REGION Network 67: FAT Mode All Check
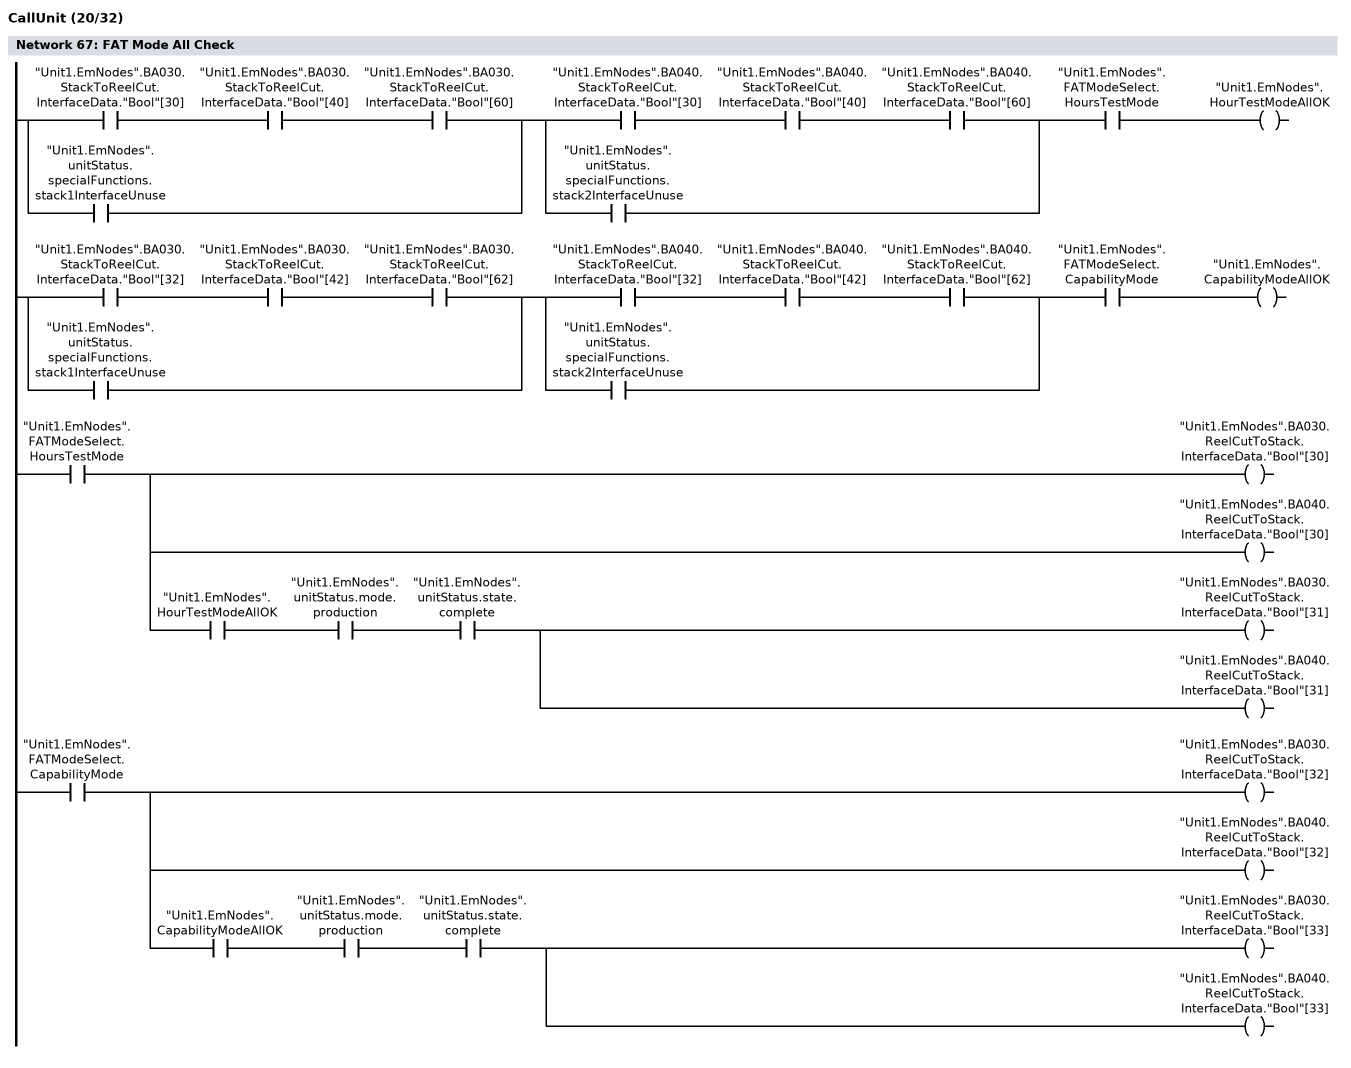
   RUNG wire#powerrail
      Contact( "Unit1.EmNodes".BA030.StackToReelCut.InterfaceData."Bool"[30] )
      Contact( "Unit1.EmNodes".BA030.StackToReelCut.InterfaceData."Bool"[40] )
      Contact( "Unit1.EmNodes".BA030.StackToReelCut.InterfaceData."Bool"[60] )
      wire#w1
      Contact( "Unit1.EmNodes".BA040.StackToReelCut.InterfaceData."Bool"[30] )
      Contact( "Unit1.EmNodes".BA040.StackToReelCut.InterfaceData."Bool"[40] )
      Contact( "Unit1.EmNodes".BA040.StackToReelCut.InterfaceData."Bool"[60] )
      wire#w2
      Contact( "Unit1.EmNodes".FATModeSelect.HoursTestMode )
      Coil( "Unit1.EmNodes".HourTestModeAllOK )
   END_RUNG
   RUNG wire#powerrail
      Contact( "Unit1.EmNodes".unitStatus.specialFunctions.stack1InterfaceUnuse )
   END_RUNG wire#w1
   RUNG wire#w1
      Contact( "Unit1.EmNodes".unitStatus.specialFunctions.stack2InterfaceUnuse )
   END_RUNG wire#w2
   RUNG wire#powerrail
      Contact( "Unit1.EmNodes".BA030.StackToReelCut.InterfaceData."Bool"[32] )
      Contact( "Unit1.EmNodes".BA030.StackToReelCut.InterfaceData."Bool"[42] )
      Contact( "Unit1.EmNodes".BA030.StackToReelCut.InterfaceData."Bool"[62] )
      wire#w3
      Contact( "Unit1.EmNodes".BA040.StackToReelCut.InterfaceData."Bool"[32] )
      Contact( "Unit1.EmNodes".BA040.StackToReelCut.InterfaceData."Bool"[42] )
      Contact( "Unit1.EmNodes".BA040.StackToReelCut.InterfaceData."Bool"[62] )
      wire#w4
      Contact( "Unit1.EmNodes".FATModeSelect.CapabilityMode )
      Coil( "Unit1.EmNodes".CapabilityModeAllOK )
   END_RUNG
   RUNG wire#powerrail
      Contact( "Unit1.EmNodes".unitStatus.specialFunctions.stack1InterfaceUnuse )
   END_RUNG wire#w3
   RUNG wire#w3
      Contact( "Unit1.EmNodes".unitStatus.specialFunctions.stack2InterfaceUnuse )
   END_RUNG wire#w4
   RUNG wire#powerrail
      Contact( "Unit1.EmNodes".FATModeSelect.HoursTestMode )
      wire#w5
      Coil( "Unit1.EmNodes".BA030.ReelCutToStack.InterfaceData."Bool"[30] )
   END_RUNG
   RUNG wire#w5
      Coil( "Unit1.EmNodes".BA040.ReelCutToStack.InterfaceData."Bool"[30] )
   END_RUNG
   RUNG wire#w5
      Contact( "Unit1.EmNodes".HourTestModeAllOK )
      Contact( "Unit1.EmNodes".unitStatus.mode.production )
      Contact( "Unit1.EmNodes".unitStatus.state.complete )
      wire#w6
      Coil( "Unit1.EmNodes".BA030.ReelCutToStack.InterfaceData."Bool"[31] )
   END_RUNG
   RUNG wire#w6
      Coil( "Unit1.EmNodes".BA040.ReelCutToStack.InterfaceData."Bool"[31] )
   END_RUNG
   RUNG wire#powerrail
      Contact( "Unit1.EmNodes".FATModeSelect.CapabilityMode )
      wire#w7
      Coil( "Unit1.EmNodes".BA030.ReelCutToStack.InterfaceData."Bool"[32] )
   END_RUNG
   RUNG wire#w7
      Coil( "Unit1.EmNodes".BA040.ReelCutToStack.InterfaceData."Bool"[32] )
   END_RUNG
   RUNG wire#w7
      Contact( "Unit1.EmNodes".CapabilityModeAllOK )
      Contact( "Unit1.EmNodes".unitStatus.mode.production )
      Contact( "Unit1.EmNodes".unitStatus.state.complete )
      wire#w8
      Coil( "Unit1.EmNodes".BA030.ReelCutToStack.InterfaceData."Bool"[33] )
   END_RUNG
   RUNG wire#w8
      Coil( "Unit1.EmNodes".BA040.ReelCutToStack.InterfaceData."Bool"[33] )
   END_RUNG
   // the same network as SCL:
   "Unit1.EmNodes".HourTestModeAllOK := (("Unit1.EmNodes".BA030.StackToReelCut.InterfaceData."Bool"[30] AND "Unit1.EmNodes".BA030.StackToReelCut.InterfaceData."Bool"[40] AND "Unit1.EmNodes".BA030.StackToReelCut.InterfaceData."Bool"[60]) OR "Unit1.EmNodes".unitStatus.specialFunctions.stack1InterfaceUnuse) AND (("Unit1.EmNodes".BA040.StackToReelCut.InterfaceData."Bool"[30] AND "Unit1.EmNodes".BA040.StackToReelCut.InterfaceData."Bool"[40] AND "Unit1.EmNodes".BA040.StackToReelCut.InterfaceData."Bool"[60]) OR "Unit1.EmNodes".unitStatus.specialFunctions.stack2InterfaceUnuse) AND "Unit1.EmNodes".FATModeSelect.HoursTestMode;
   "Unit1.EmNodes".CapabilityModeAllOK := (("Unit1.EmNodes".BA030.StackToReelCut.InterfaceData."Bool"[32] AND "Unit1.EmNodes".BA030.StackToReelCut.InterfaceData."Bool"[42] AND "Unit1.EmNodes".BA030.StackToReelCut.InterfaceData."Bool"[62]) OR "Unit1.EmNodes".unitStatus.specialFunctions.stack1InterfaceUnuse) AND (("Unit1.EmNodes".BA040.StackToReelCut.InterfaceData."Bool"[32] AND "Unit1.EmNodes".BA040.StackToReelCut.InterfaceData."Bool"[42] AND "Unit1.EmNodes".BA040.StackToReelCut.InterfaceData."Bool"[62]) OR "Unit1.EmNodes".unitStatus.specialFunctions.stack2InterfaceUnuse) AND "Unit1.EmNodes".FATModeSelect.CapabilityMode;
   "Unit1.EmNodes".BA030.ReelCutToStack.InterfaceData."Bool"[30] := "Unit1.EmNodes".FATModeSelect.HoursTestMode;
   "Unit1.EmNodes".BA040.ReelCutToStack.InterfaceData."Bool"[30] := "Unit1.EmNodes".FATModeSelect.HoursTestMode;
   "Unit1.EmNodes".BA030.ReelCutToStack.InterfaceData."Bool"[31] := "Unit1.EmNodes".FATModeSelect.HoursTestMode AND "Unit1.EmNodes".HourTestModeAllOK AND "Unit1.EmNodes".unitStatus.mode.production AND "Unit1.EmNodes".unitStatus.state.complete;
   "Unit1.EmNodes".BA040.ReelCutToStack.InterfaceData."Bool"[31] := "Unit1.EmNodes".FATModeSelect.HoursTestMode AND "Unit1.EmNodes".HourTestModeAllOK AND "Unit1.EmNodes".unitStatus.mode.production AND "Unit1.EmNodes".unitStatus.state.complete;
   "Unit1.EmNodes".BA030.ReelCutToStack.InterfaceData."Bool"[32] := "Unit1.EmNodes".FATModeSelect.CapabilityMode;
   "Unit1.EmNodes".BA040.ReelCutToStack.InterfaceData."Bool"[32] := "Unit1.EmNodes".FATModeSelect.CapabilityMode;
   "Unit1.EmNodes".BA030.ReelCutToStack.InterfaceData."Bool"[33] := "Unit1.EmNodes".FATModeSelect.CapabilityMode AND "Unit1.EmNodes".CapabilityModeAllOK AND "Unit1.EmNodes".unitStatus.mode.production AND "Unit1.EmNodes".unitStatus.state.complete;
   "Unit1.EmNodes".BA040.ReelCutToStack.InterfaceData."Bool"[33] := "Unit1.EmNodes".FATModeSelect.CapabilityMode AND "Unit1.EmNodes".CapabilityModeAllOK AND "Unit1.EmNodes".unitStatus.mode.production AND "Unit1.EmNodes".unitStatus.state.complete;
END_REGION

REGION Network 68: HoursTest Mode
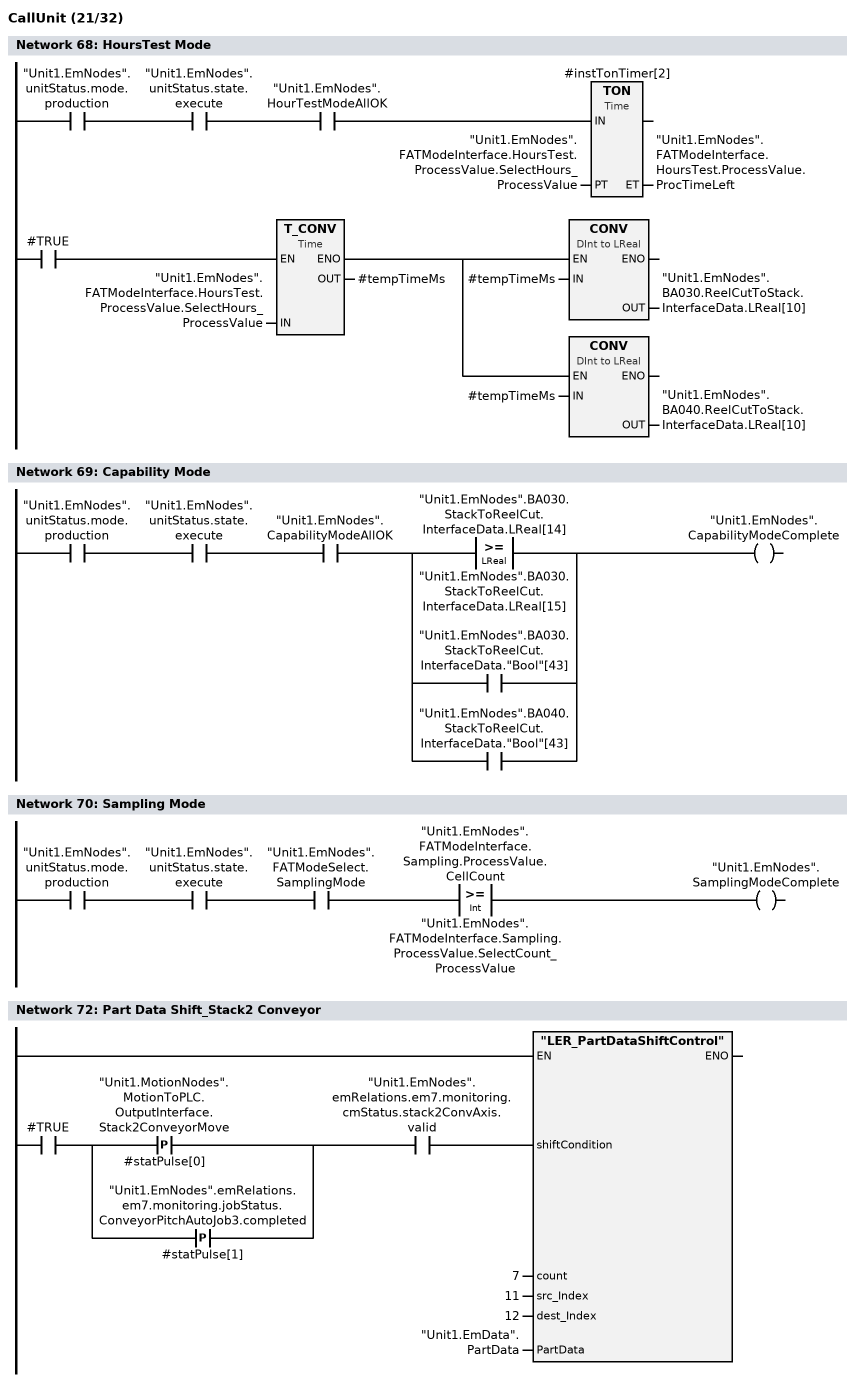
   RUNG wire#powerrail
      Contact( "Unit1.EmNodes".unitStatus.mode.production )
      Contact( "Unit1.EmNodes".unitStatus.state.execute )
      Contact( "Unit1.EmNodes".HourTestModeAllOK )
      { S7_Templates := "time_type := Time" } #instTonTimer[2].TON(pt := "Unit1.EmNodes".FATModeInterface.HoursTest.ProcessValue.SelectHours_ProcessValue, et => "Unit1.EmNodes".FATModeInterface.HoursTest.ProcessValue.ProcTimeLeft)
   END_RUNG
   RUNG wire#powerrail
      Contact( #TRUE )
      { S7_Templates := "[src_type := Time, dest_type := DInt]" } T_CONV(IN := "Unit1.EmNodes".FATModeInterface.HoursTest.ProcessValue.SelectHours_ProcessValue, OUT => #tempTimeMs)
      wire#w1
      { S7_Templates := "[SrcType := DInt, DestType := LReal]" } Convert(in := #tempTimeMs, out => "Unit1.EmNodes".BA030.ReelCutToStack.InterfaceData.LReal[10])
   END_RUNG
   RUNG wire#w1
      { S7_Templates := "[SrcType := DInt, DestType := LReal]" } Convert(in := #tempTimeMs, out => "Unit1.EmNodes".BA040.ReelCutToStack.InterfaceData.LReal[10])
   END_RUNG
   // the same network as SCL:
   #instTonTimer[2].TON(IN := "Unit1.EmNodes".unitStatus.mode.production AND "Unit1.EmNodes".unitStatus.state.execute AND "Unit1.EmNodes".HourTestModeAllOK,
                        PT := "Unit1.EmNodes".FATModeInterface.HoursTest.ProcessValue.SelectHours_ProcessValue,
                        ET => "Unit1.EmNodes".FATModeInterface.HoursTest.ProcessValue.ProcTimeLeft);
   T_CONV(EN := #TRUE,
          IN := "Unit1.EmNodes".FATModeInterface.HoursTest.ProcessValue.SelectHours_ProcessValue,
          OUT => #tempTimeMs,
          ENO => #_w1);
   IF #_w1 THEN
       "Unit1.EmNodes".BA030.ReelCutToStack.InterfaceData.LReal[10] := DINT_TO_LREAL(#tempTimeMs);
       "Unit1.EmNodes".BA040.ReelCutToStack.InterfaceData.LReal[10] := DINT_TO_LREAL(#tempTimeMs);
   END_IF;
END_REGION

REGION Network 69: Capability Mode
   RUNG wire#powerrail
      Contact( "Unit1.EmNodes".unitStatus.mode.production )
      Contact( "Unit1.EmNodes".unitStatus.state.execute )
      Contact( "Unit1.EmNodes".CapabilityModeAllOK )
      wire#w1
      { S7_Templates := "SrcType := LReal" } GE_Contact(in1 := "Unit1.EmNodes".BA030.StackToReelCut.InterfaceData.LReal[14], in2 := "Unit1.EmNodes".BA030.StackToReelCut.InterfaceData.LReal[15])
      wire#w2
      Coil( "Unit1.EmNodes".CapabilityModeComplete )
   END_RUNG
   RUNG wire#w1
      Contact( "Unit1.EmNodes".BA030.StackToReelCut.InterfaceData."Bool"[43] )
   END_RUNG wire#w2
   RUNG wire#w1
      Contact( "Unit1.EmNodes".BA040.StackToReelCut.InterfaceData."Bool"[43] )
   END_RUNG wire#w2
   // the same network as SCL:
   "Unit1.EmNodes".CapabilityModeComplete := "Unit1.EmNodes".unitStatus.mode.production AND "Unit1.EmNodes".unitStatus.state.execute AND "Unit1.EmNodes".CapabilityModeAllOK AND (("Unit1.EmNodes".BA030.StackToReelCut.InterfaceData.LReal[14] >= "Unit1.EmNodes".BA030.StackToReelCut.InterfaceData.LReal[15]) OR "Unit1.EmNodes".BA030.StackToReelCut.InterfaceData."Bool"[43] OR "Unit1.EmNodes".BA040.StackToReelCut.InterfaceData."Bool"[43]);
END_REGION

REGION Network 70: Sampling Mode
   RUNG wire#powerrail
      Contact( "Unit1.EmNodes".unitStatus.mode.production )
      Contact( "Unit1.EmNodes".unitStatus.state.execute )
      Contact( "Unit1.EmNodes".FATModeSelect.SamplingMode )
      { S7_Templates := "SrcType := Int" } GE_Contact(in1 := "Unit1.EmNodes".FATModeInterface.Sampling.ProcessValue.CellCount, in2 := "Unit1.EmNodes".FATModeInterface.Sampling.ProcessValue.SelectCount_ProcessValue)
      Coil( "Unit1.EmNodes".SamplingModeComplete )
   END_RUNG
   // the same network as SCL:
   "Unit1.EmNodes".SamplingModeComplete := "Unit1.EmNodes".unitStatus.mode.production AND "Unit1.EmNodes".unitStatus.state.execute AND "Unit1.EmNodes".FATModeSelect.SamplingMode AND ("Unit1.EmNodes".FATModeInterface.Sampling.ProcessValue.CellCount >= "Unit1.EmNodes".FATModeInterface.Sampling.ProcessValue.SelectCount_ProcessValue);
END_REGION

REGION Network 71: ******************** Part Data Shift ********************
END_REGION

REGION Network 72: Part Data Shift_Stack2 Conveyor
   RUNG wire#powerrail
      "LER_PartDataShiftControl"(shiftCondition := wire#w3, count := 7, src_Index := 11, dest_Index := 12, PartData := "Unit1.EmData".PartData)
   END_RUNG
   RUNG wire#powerrail
      Contact( #TRUE )
      wire#w1
      P_Contact(operand := "Unit1.MotionNodes".MotionToPLC.OutputInterface.Stack2ConveyorMove, bit := #statPulse[0])
      wire#w2
      Contact( "Unit1.EmNodes".emRelations.em7.monitoring.cmStatus.stack2ConvAxis.valid )
   END_RUNG wire#w3
   RUNG wire#w1
      P_Contact(operand := "Unit1.EmNodes".emRelations.em7.monitoring.jobStatus.ConveyorPitchAutoJob3.completed, bit := #statPulse[1])
   END_RUNG wire#w2
   // the same network as SCL:
   #_w1 := #TRUE AND "Unit1.MotionNodes".MotionToPLC.OutputInterface.Stack2ConveyorMove AND NOT #statPulse[0];   // rising edge of "Unit1.MotionNodes".MotionToPLC.OutputInterface.Stack2ConveyorMove
   #statPulse[0] := "Unit1.MotionNodes".MotionToPLC.OutputInterface.Stack2ConveyorMove;
   #_w2 := #TRUE AND "Unit1.EmNodes".emRelations.em7.monitoring.jobStatus.ConveyorPitchAutoJob3.completed AND NOT #statPulse[1];   // rising edge of "Unit1.EmNodes".emRelations.em7.monitoring.jobStatus.ConveyorPitchAutoJob3.completed
   #statPulse[1] := "Unit1.EmNodes".emRelations.em7.monitoring.jobStatus.ConveyorPitchAutoJob3.completed;
   "LER_PartDataShiftControl"(shiftCondition := (#_w1 OR #_w2) AND "Unit1.EmNodes".emRelations.em7.monitoring.cmStatus.stack2ConvAxis.valid,
                           count := 7,
                           src_Index := 11,
                           dest_Index := 12,
                           PartData := "Unit1.EmData".PartData);
END_REGION

REGION Network 73: Part Data Shift_Stack1 Conveyor
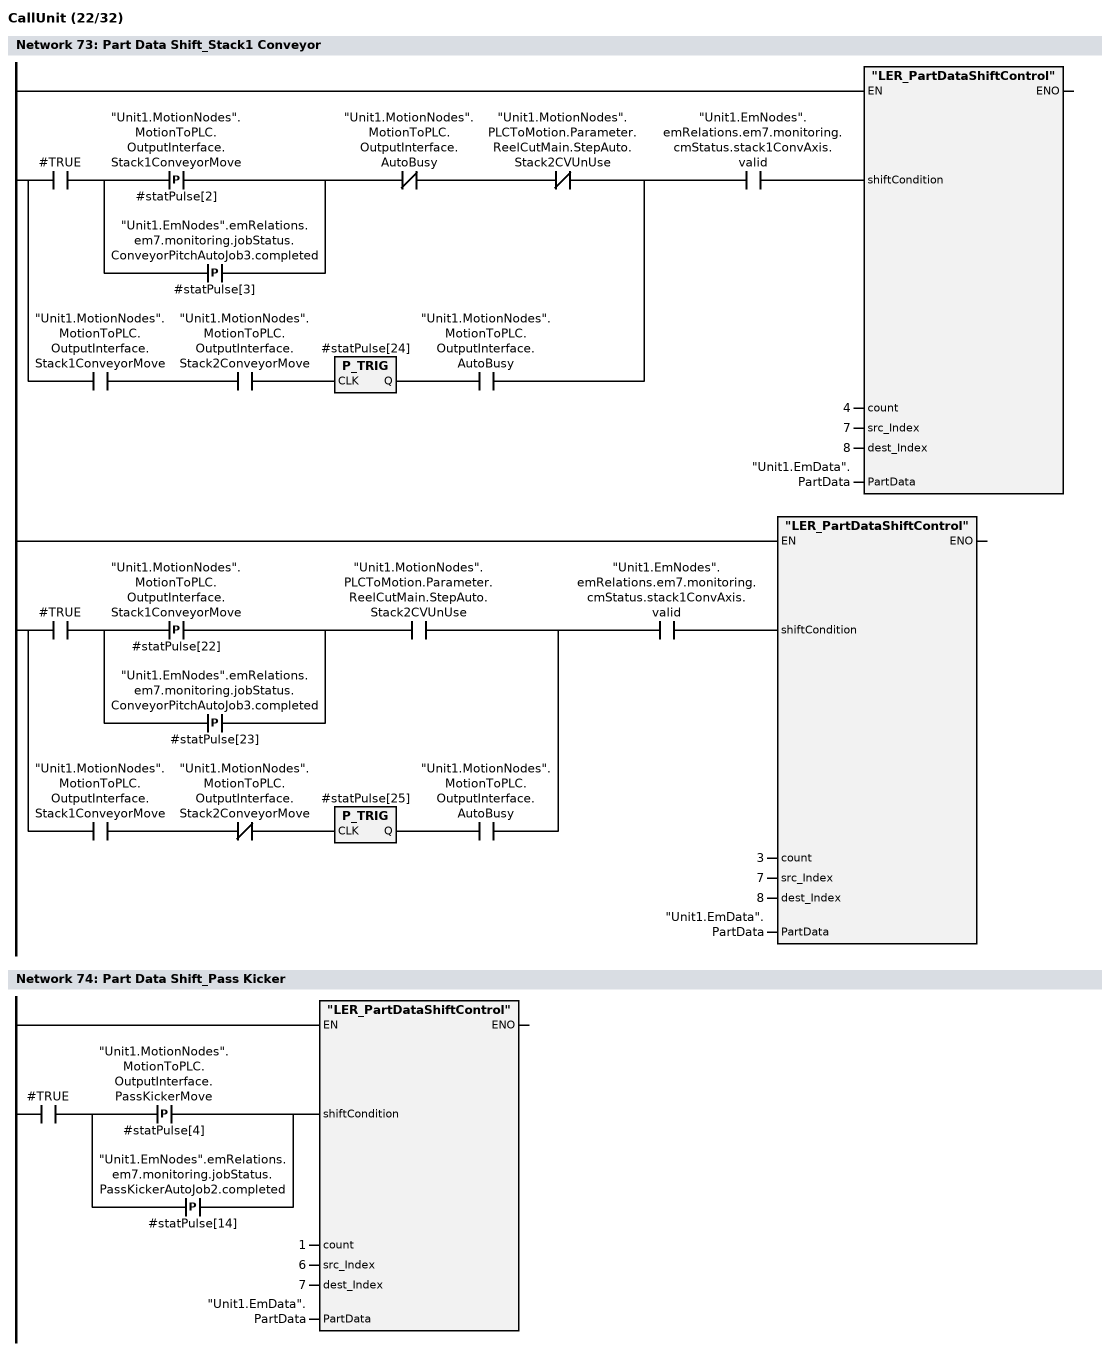
   RUNG wire#powerrail
      "LER_PartDataShiftControl"(shiftCondition := wire#w4, count := 4, src_Index := 7, dest_Index := 8, PartData := "Unit1.EmData".PartData)
   END_RUNG
   RUNG wire#powerrail
      Contact( #TRUE )
      wire#w1
      P_Contact(operand := "Unit1.MotionNodes".MotionToPLC.OutputInterface.Stack1ConveyorMove, bit := #statPulse[2])
      wire#w2
      I_Contact( "Unit1.MotionNodes".MotionToPLC.OutputInterface.AutoBusy )
      I_Contact( "Unit1.MotionNodes".PLCToMotion.Parameter.ReelCutMain.StepAuto.Stack2CVUnUse )
      wire#w3
      Contact( "Unit1.EmNodes".emRelations.em7.monitoring.cmStatus.stack1ConvAxis.valid )
   END_RUNG wire#w4
   RUNG wire#w1
      P_Contact(operand := "Unit1.EmNodes".emRelations.em7.monitoring.jobStatus.ConveyorPitchAutoJob3.completed, bit := #statPulse[3])
   END_RUNG wire#w2
   RUNG wire#powerrail
      Contact( "Unit1.MotionNodes".MotionToPLC.OutputInterface.Stack1ConveyorMove )
      Contact( "Unit1.MotionNodes".MotionToPLC.OutputInterface.Stack2ConveyorMove )
      P_Trig( #statPulse[24] )
      Contact( "Unit1.MotionNodes".MotionToPLC.OutputInterface.AutoBusy )
   END_RUNG wire#w3
   RUNG wire#powerrail
      "LER_PartDataShiftControl"(shiftCondition := wire#w8, count := 3, src_Index := 7, dest_Index := 8, PartData := "Unit1.EmData".PartData)
   END_RUNG
   RUNG wire#powerrail
      Contact( #TRUE )
      wire#w5
      P_Contact(operand := "Unit1.MotionNodes".MotionToPLC.OutputInterface.Stack1ConveyorMove, bit := #statPulse[22])
      wire#w6
      Contact( "Unit1.MotionNodes".PLCToMotion.Parameter.ReelCutMain.StepAuto.Stack2CVUnUse )
      wire#w7
      Contact( "Unit1.EmNodes".emRelations.em7.monitoring.cmStatus.stack1ConvAxis.valid )
   END_RUNG wire#w8
   RUNG wire#w5
      P_Contact(operand := "Unit1.EmNodes".emRelations.em7.monitoring.jobStatus.ConveyorPitchAutoJob3.completed, bit := #statPulse[23])
   END_RUNG wire#w6
   RUNG wire#powerrail
      Contact( "Unit1.MotionNodes".MotionToPLC.OutputInterface.Stack1ConveyorMove )
      I_Contact( "Unit1.MotionNodes".MotionToPLC.OutputInterface.Stack2ConveyorMove )
      P_Trig( #statPulse[25] )
      Contact( "Unit1.MotionNodes".MotionToPLC.OutputInterface.AutoBusy )
   END_RUNG wire#w7
   // the same network as SCL:
   #_w1 := #TRUE AND "Unit1.MotionNodes".MotionToPLC.OutputInterface.Stack1ConveyorMove AND NOT #statPulse[2];   // rising edge of "Unit1.MotionNodes".MotionToPLC.OutputInterface.Stack1ConveyorMove
   #statPulse[2] := "Unit1.MotionNodes".MotionToPLC.OutputInterface.Stack1ConveyorMove;
   #_w2 := #TRUE AND "Unit1.EmNodes".emRelations.em7.monitoring.jobStatus.ConveyorPitchAutoJob3.completed AND NOT #statPulse[3];   // rising edge of "Unit1.EmNodes".emRelations.em7.monitoring.jobStatus.ConveyorPitchAutoJob3.completed
   #statPulse[3] := "Unit1.EmNodes".emRelations.em7.monitoring.jobStatus.ConveyorPitchAutoJob3.completed;
   #_w3 := "Unit1.MotionNodes".MotionToPLC.OutputInterface.Stack1ConveyorMove AND "Unit1.MotionNodes".MotionToPLC.OutputInterface.Stack2ConveyorMove;
   #_w4 := #_w3 AND NOT #statPulse[24];   // rising edge
   #statPulse[24] := #_w3;
   "LER_PartDataShiftControl"(shiftCondition := (((#_w1 OR #_w2) AND NOT "Unit1.MotionNodes".MotionToPLC.OutputInterface.AutoBusy AND NOT "Unit1.MotionNodes".PLCToMotion.Parameter.ReelCutMain.StepAuto.Stack2CVUnUse) OR (#_w4 AND "Unit1.MotionNodes".MotionToPLC.OutputInterface.AutoBusy)) AND "Unit1.EmNodes".emRelations.em7.monitoring.cmStatus.stack1ConvAxis.valid,
                           count := 4,
                           src_Index := 7,
                           dest_Index := 8,
                           PartData := "Unit1.EmData".PartData);
   #_w5 := #TRUE AND "Unit1.MotionNodes".MotionToPLC.OutputInterface.Stack1ConveyorMove AND NOT #statPulse[22];   // rising edge of "Unit1.MotionNodes".MotionToPLC.OutputInterface.Stack1ConveyorMove
   #statPulse[22] := "Unit1.MotionNodes".MotionToPLC.OutputInterface.Stack1ConveyorMove;
   #_w6 := #TRUE AND "Unit1.EmNodes".emRelations.em7.monitoring.jobStatus.ConveyorPitchAutoJob3.completed AND NOT #statPulse[23];   // rising edge of "Unit1.EmNodes".emRelations.em7.monitoring.jobStatus.ConveyorPitchAutoJob3.completed
   #statPulse[23] := "Unit1.EmNodes".emRelations.em7.monitoring.jobStatus.ConveyorPitchAutoJob3.completed;
   #_w7 := "Unit1.MotionNodes".MotionToPLC.OutputInterface.Stack1ConveyorMove AND NOT "Unit1.MotionNodes".MotionToPLC.OutputInterface.Stack2ConveyorMove;
   #_w8 := #_w7 AND NOT #statPulse[25];   // rising edge
   #statPulse[25] := #_w7;
   "LER_PartDataShiftControl"(shiftCondition := (((#_w5 OR #_w6) AND "Unit1.MotionNodes".PLCToMotion.Parameter.ReelCutMain.StepAuto.Stack2CVUnUse) OR (#_w8 AND "Unit1.MotionNodes".MotionToPLC.OutputInterface.AutoBusy)) AND "Unit1.EmNodes".emRelations.em7.monitoring.cmStatus.stack1ConvAxis.valid,
                           count := 3,
                           src_Index := 7,
                           dest_Index := 8,
                           PartData := "Unit1.EmData".PartData);
END_REGION

REGION Network 74: Part Data Shift_Pass Kicker
   RUNG wire#powerrail
      "LER_PartDataShiftControl"(shiftCondition := wire#w2, count := 1, src_Index := 6, dest_Index := 7, PartData := "Unit1.EmData".PartData)
   END_RUNG
   RUNG wire#powerrail
      Contact( #TRUE )
      wire#w1
      P_Contact(operand := "Unit1.MotionNodes".MotionToPLC.OutputInterface.PassKickerMove, bit := #statPulse[4])
   END_RUNG wire#w2
   RUNG wire#w1
      P_Contact(operand := "Unit1.EmNodes".emRelations.em7.monitoring.jobStatus.PassKickerAutoJob2.completed, bit := #statPulse[14])
   END_RUNG wire#w2
   // the same network as SCL:
   #_w1 := #TRUE AND "Unit1.MotionNodes".MotionToPLC.OutputInterface.PassKickerMove AND NOT #statPulse[4];   // rising edge of "Unit1.MotionNodes".MotionToPLC.OutputInterface.PassKickerMove
   #statPulse[4] := "Unit1.MotionNodes".MotionToPLC.OutputInterface.PassKickerMove;
   #_w2 := #TRUE AND "Unit1.EmNodes".emRelations.em7.monitoring.jobStatus.PassKickerAutoJob2.completed AND NOT #statPulse[14];   // rising edge of "Unit1.EmNodes".emRelations.em7.monitoring.jobStatus.PassKickerAutoJob2.completed
   #statPulse[14] := "Unit1.EmNodes".emRelations.em7.monitoring.jobStatus.PassKickerAutoJob2.completed;
   "LER_PartDataShiftControl"(shiftCondition := #_w1 OR #_w2,
                           count := 1,
                           src_Index := 6,
                           dest_Index := 7,
                           PartData := "Unit1.EmData".PartData);
END_REGION

REGION Network 75: Part Data Shift_NG Kicker
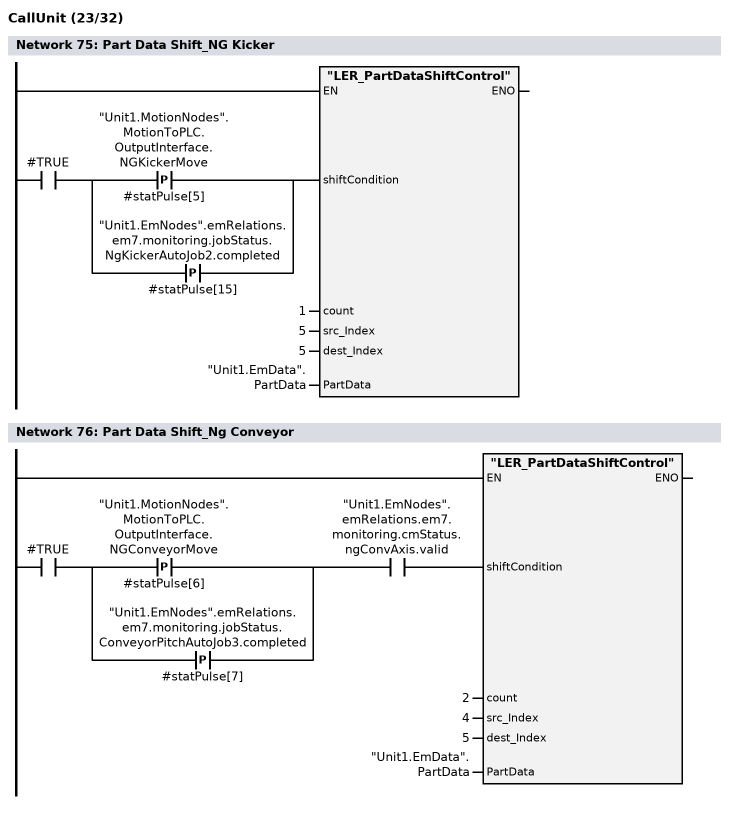
   RUNG wire#powerrail
      "LER_PartDataShiftControl"(shiftCondition := wire#w2, count := 1, src_Index := 5, dest_Index := 5, PartData := "Unit1.EmData".PartData)
   END_RUNG
   RUNG wire#powerrail
      Contact( #TRUE )
      wire#w1
      P_Contact(operand := "Unit1.MotionNodes".MotionToPLC.OutputInterface.NGKickerMove, bit := #statPulse[5])
   END_RUNG wire#w2
   RUNG wire#w1
      P_Contact(operand := "Unit1.EmNodes".emRelations.em7.monitoring.jobStatus.NgKickerAutoJob2.completed, bit := #statPulse[15])
   END_RUNG wire#w2
   // the same network as SCL:
   #_w1 := #TRUE AND "Unit1.MotionNodes".MotionToPLC.OutputInterface.NGKickerMove AND NOT #statPulse[5];   // rising edge of "Unit1.MotionNodes".MotionToPLC.OutputInterface.NGKickerMove
   #statPulse[5] := "Unit1.MotionNodes".MotionToPLC.OutputInterface.NGKickerMove;
   #_w2 := #TRUE AND "Unit1.EmNodes".emRelations.em7.monitoring.jobStatus.NgKickerAutoJob2.completed AND NOT #statPulse[15];   // rising edge of "Unit1.EmNodes".emRelations.em7.monitoring.jobStatus.NgKickerAutoJob2.completed
   #statPulse[15] := "Unit1.EmNodes".emRelations.em7.monitoring.jobStatus.NgKickerAutoJob2.completed;
   "LER_PartDataShiftControl"(shiftCondition := #_w1 OR #_w2,
                           count := 1,
                           src_Index := 5,
                           dest_Index := 5,
                           PartData := "Unit1.EmData".PartData);
END_REGION

REGION Network 76: Part Data Shift_Ng Conveyor
   RUNG wire#powerrail
      "LER_PartDataShiftControl"(shiftCondition := wire#w3, count := 2, src_Index := 4, dest_Index := 5, PartData := "Unit1.EmData".PartData)
   END_RUNG
   RUNG wire#powerrail
      Contact( #TRUE )
      wire#w1
      P_Contact(operand := "Unit1.MotionNodes".MotionToPLC.OutputInterface.NGConveyorMove, bit := #statPulse[6])
      wire#w2
      Contact( "Unit1.EmNodes".emRelations.em7.monitoring.cmStatus.ngConvAxis.valid )
   END_RUNG wire#w3
   RUNG wire#w1
      P_Contact(operand := "Unit1.EmNodes".emRelations.em7.monitoring.jobStatus.ConveyorPitchAutoJob3.completed, bit := #statPulse[7])
   END_RUNG wire#w2
   // the same network as SCL:
   #_w1 := #TRUE AND "Unit1.MotionNodes".MotionToPLC.OutputInterface.NGConveyorMove AND NOT #statPulse[6];   // rising edge of "Unit1.MotionNodes".MotionToPLC.OutputInterface.NGConveyorMove
   #statPulse[6] := "Unit1.MotionNodes".MotionToPLC.OutputInterface.NGConveyorMove;
   #_w2 := #TRUE AND "Unit1.EmNodes".emRelations.em7.monitoring.jobStatus.ConveyorPitchAutoJob3.completed AND NOT #statPulse[7];   // rising edge of "Unit1.EmNodes".emRelations.em7.monitoring.jobStatus.ConveyorPitchAutoJob3.completed
   #statPulse[7] := "Unit1.EmNodes".emRelations.em7.monitoring.jobStatus.ConveyorPitchAutoJob3.completed;
   "LER_PartDataShiftControl"(shiftCondition := (#_w1 OR #_w2) AND "Unit1.EmNodes".emRelations.em7.monitoring.cmStatus.ngConvAxis.valid,
                           count := 2,
                           src_Index := 4,
                           dest_Index := 5,
                           PartData := "Unit1.EmData".PartData);
END_REGION

REGION Network 77: Part Data Shift_Cut Conveyor
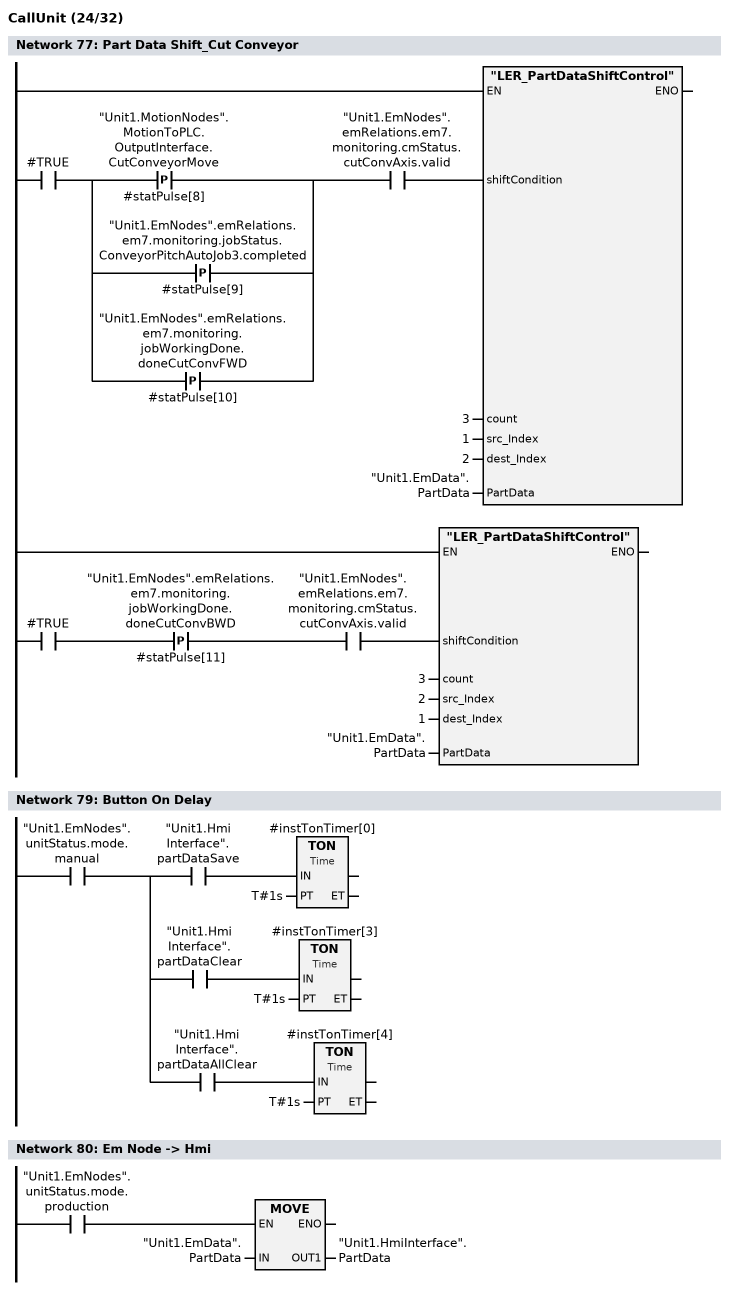
   RUNG wire#powerrail
      "LER_PartDataShiftControl"(shiftCondition := wire#w3, count := 3, src_Index := 1, dest_Index := 2, PartData := "Unit1.EmData".PartData)
   END_RUNG
   RUNG wire#powerrail
      Contact( #TRUE )
      wire#w1
      P_Contact(operand := "Unit1.MotionNodes".MotionToPLC.OutputInterface.CutConveyorMove, bit := #statPulse[8])
      wire#w2
      Contact( "Unit1.EmNodes".emRelations.em7.monitoring.cmStatus.cutConvAxis.valid )
   END_RUNG wire#w3
   RUNG wire#w1
      P_Contact(operand := "Unit1.EmNodes".emRelations.em7.monitoring.jobStatus.ConveyorPitchAutoJob3.completed, bit := #statPulse[9])
   END_RUNG wire#w2
   RUNG wire#w1
      P_Contact(operand := "Unit1.EmNodes".emRelations.em7.monitoring.jobWorkingDone.doneCutConvFWD, bit := #statPulse[10])
   END_RUNG wire#w2
   RUNG wire#powerrail
      "LER_PartDataShiftControl"(shiftCondition := wire#w4, count := 3, src_Index := 2, dest_Index := 1, PartData := "Unit1.EmData".PartData)
   END_RUNG
   RUNG wire#powerrail
      Contact( #TRUE )
      P_Contact(operand := "Unit1.EmNodes".emRelations.em7.monitoring.jobWorkingDone.doneCutConvBWD, bit := #statPulse[11])
      Contact( "Unit1.EmNodes".emRelations.em7.monitoring.cmStatus.cutConvAxis.valid )
   END_RUNG wire#w4
   // the same network as SCL:
   #_w1 := #TRUE AND "Unit1.MotionNodes".MotionToPLC.OutputInterface.CutConveyorMove AND NOT #statPulse[8];   // rising edge of "Unit1.MotionNodes".MotionToPLC.OutputInterface.CutConveyorMove
   #statPulse[8] := "Unit1.MotionNodes".MotionToPLC.OutputInterface.CutConveyorMove;
   #_w2 := #TRUE AND "Unit1.EmNodes".emRelations.em7.monitoring.jobStatus.ConveyorPitchAutoJob3.completed AND NOT #statPulse[9];   // rising edge of "Unit1.EmNodes".emRelations.em7.monitoring.jobStatus.ConveyorPitchAutoJob3.completed
   #statPulse[9] := "Unit1.EmNodes".emRelations.em7.monitoring.jobStatus.ConveyorPitchAutoJob3.completed;
   #_w3 := #TRUE AND "Unit1.EmNodes".emRelations.em7.monitoring.jobWorkingDone.doneCutConvFWD AND NOT #statPulse[10];   // rising edge of "Unit1.EmNodes".emRelations.em7.monitoring.jobWorkingDone.doneCutConvFWD
   #statPulse[10] := "Unit1.EmNodes".emRelations.em7.monitoring.jobWorkingDone.doneCutConvFWD;
   "LER_PartDataShiftControl"(shiftCondition := (#_w1 OR #_w2 OR #_w3) AND "Unit1.EmNodes".emRelations.em7.monitoring.cmStatus.cutConvAxis.valid,
                           count := 3,
                           src_Index := 1,
                           dest_Index := 2,
                           PartData := "Unit1.EmData".PartData);
   #_w4 := #TRUE AND "Unit1.EmNodes".emRelations.em7.monitoring.jobWorkingDone.doneCutConvBWD AND NOT #statPulse[11];   // rising edge of "Unit1.EmNodes".emRelations.em7.monitoring.jobWorkingDone.doneCutConvBWD
   #statPulse[11] := "Unit1.EmNodes".emRelations.em7.monitoring.jobWorkingDone.doneCutConvBWD;
   "LER_PartDataShiftControl"(shiftCondition := #_w4 AND "Unit1.EmNodes".emRelations.em7.monitoring.cmStatus.cutConvAxis.valid,
                           count := 3,
                           src_Index := 2,
                           dest_Index := 1,
                           PartData := "Unit1.EmData".PartData);
END_REGION

REGION Network 78: ==================== DATA OPERATING ======================
END_REGION

REGION Network 79: Button On Delay
   RUNG wire#powerrail
      Contact( "Unit1.EmNodes".unitStatus.mode.manual )
      wire#w1
      Contact( "Unit1.HmiInterface".partDataSave )
      { S7_Templates := "time_type := Time" } #instTonTimer[0].TON(pt := T#1s, et =>)
   END_RUNG
   RUNG wire#w1
      Contact( "Unit1.HmiInterface".partDataClear )
      { S7_Templates := "time_type := Time" } #instTonTimer[3].TON(pt := T#1s, et =>)
   END_RUNG
   RUNG wire#w1
      Contact( "Unit1.HmiInterface".partDataAllClear )
      { S7_Templates := "time_type := Time" } #instTonTimer[4].TON(pt := T#1s, et =>)
   END_RUNG
   // the same network as SCL:
   #instTonTimer[0].TON(IN := "Unit1.EmNodes".unitStatus.mode.manual AND "Unit1.HmiInterface".partDataSave,
                        PT := T#1s);
   #instTonTimer[3].TON(IN := "Unit1.EmNodes".unitStatus.mode.manual AND "Unit1.HmiInterface".partDataClear,
                        PT := T#1s);
   #instTonTimer[4].TON(IN := "Unit1.EmNodes".unitStatus.mode.manual AND "Unit1.HmiInterface".partDataAllClear,
                        PT := T#1s);
END_REGION

REGION Network 80: Em Node -> Hmi
   RUNG wire#powerrail
      Contact( "Unit1.EmNodes".unitStatus.mode.production )
      Move(in := "Unit1.EmData".PartData, out1 => "Unit1.HmiInterface".PartData)
   END_RUNG
   // the same network as SCL:
   IF "Unit1.EmNodes".unitStatus.mode.production THEN
       "Unit1.HmiInterface".PartData := "Unit1.EmData".PartData;
   END_IF;
END_REGION

REGION Network 81: Save Command HMI -> Em Node
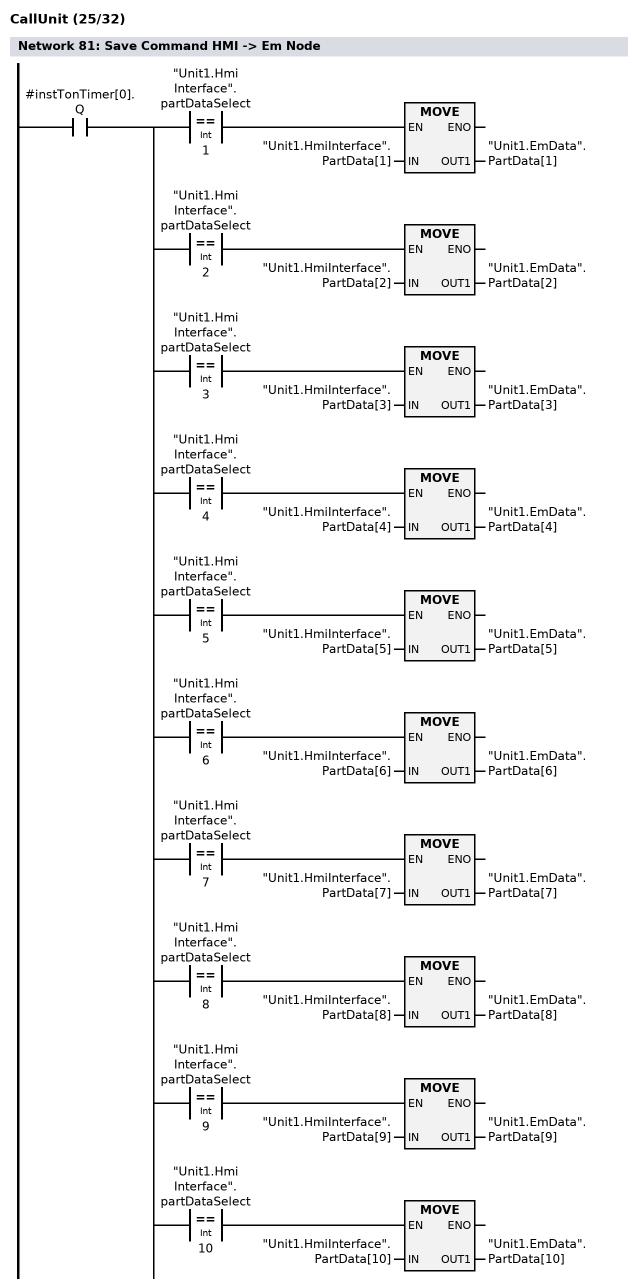
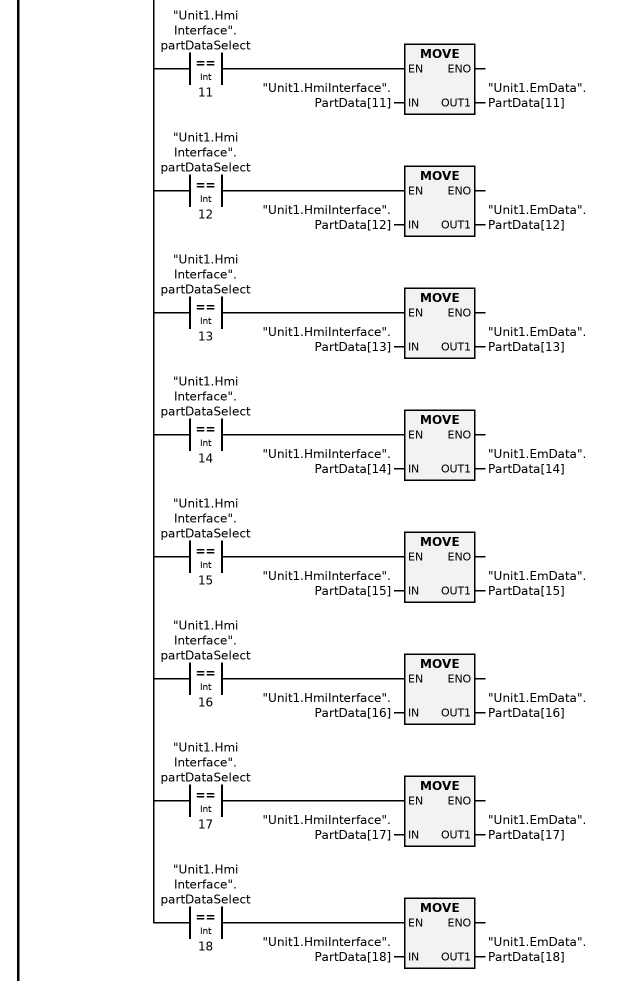
   RUNG wire#powerrail
      Contact( #instTonTimer[0].Q )
      wire#w1
      { S7_Templates := "SrcType := Int" } EQ_Contact(in1 := "Unit1.HmiInterface".partDataSelect, in2 := 1)
      Move(in := "Unit1.HmiInterface".PartData[1], out1 => "Unit1.EmData".PartData[1])
   END_RUNG
   RUNG wire#w1
      { S7_Templates := "SrcType := Int" } EQ_Contact(in1 := "Unit1.HmiInterface".partDataSelect, in2 := 2)
      Move(in := "Unit1.HmiInterface".PartData[2], out1 => "Unit1.EmData".PartData[2])
   END_RUNG
   RUNG wire#w1
      { S7_Templates := "SrcType := Int" } EQ_Contact(in1 := "Unit1.HmiInterface".partDataSelect, in2 := 3)
      Move(in := "Unit1.HmiInterface".PartData[3], out1 => "Unit1.EmData".PartData[3])
   END_RUNG
   RUNG wire#w1
      { S7_Templates := "SrcType := Int" } EQ_Contact(in1 := "Unit1.HmiInterface".partDataSelect, in2 := 4)
      Move(in := "Unit1.HmiInterface".PartData[4], out1 => "Unit1.EmData".PartData[4])
   END_RUNG
   RUNG wire#w1
      { S7_Templates := "SrcType := Int" } EQ_Contact(in1 := "Unit1.HmiInterface".partDataSelect, in2 := 5)
      Move(in := "Unit1.HmiInterface".PartData[5], out1 => "Unit1.EmData".PartData[5])
   END_RUNG
   RUNG wire#w1
      { S7_Templates := "SrcType := Int" } EQ_Contact(in1 := "Unit1.HmiInterface".partDataSelect, in2 := 6)
      Move(in := "Unit1.HmiInterface".PartData[6], out1 => "Unit1.EmData".PartData[6])
   END_RUNG
   RUNG wire#w1
      { S7_Templates := "SrcType := Int" } EQ_Contact(in1 := "Unit1.HmiInterface".partDataSelect, in2 := 7)
      Move(in := "Unit1.HmiInterface".PartData[7], out1 => "Unit1.EmData".PartData[7])
   END_RUNG
   RUNG wire#w1
      { S7_Templates := "SrcType := Int" } EQ_Contact(in1 := "Unit1.HmiInterface".partDataSelect, in2 := 8)
      Move(in := "Unit1.HmiInterface".PartData[8], out1 => "Unit1.EmData".PartData[8])
   END_RUNG
   RUNG wire#w1
      { S7_Templates := "SrcType := Int" } EQ_Contact(in1 := "Unit1.HmiInterface".partDataSelect, in2 := 9)
      Move(in := "Unit1.HmiInterface".PartData[9], out1 => "Unit1.EmData".PartData[9])
   END_RUNG
   RUNG wire#w1
      { S7_Templates := "SrcType := Int" } EQ_Contact(in1 := "Unit1.HmiInterface".partDataSelect, in2 := 10)
      Move(in := "Unit1.HmiInterface".PartData[10], out1 => "Unit1.EmData".PartData[10])
   END_RUNG
   RUNG wire#w1
      { S7_Templates := "SrcType := Int" } EQ_Contact(in1 := "Unit1.HmiInterface".partDataSelect, in2 := 11)
      Move(in := "Unit1.HmiInterface".PartData[11], out1 => "Unit1.EmData".PartData[11])
   END_RUNG
   RUNG wire#w1
      { S7_Templates := "SrcType := Int" } EQ_Contact(in1 := "Unit1.HmiInterface".partDataSelect, in2 := 12)
      Move(in := "Unit1.HmiInterface".PartData[12], out1 => "Unit1.EmData".PartData[12])
   END_RUNG
   RUNG wire#w1
      { S7_Templates := "SrcType := Int" } EQ_Contact(in1 := "Unit1.HmiInterface".partDataSelect, in2 := 13)
      Move(in := "Unit1.HmiInterface".PartData[13], out1 => "Unit1.EmData".PartData[13])
   END_RUNG
   RUNG wire#w1
      { S7_Templates := "SrcType := Int" } EQ_Contact(in1 := "Unit1.HmiInterface".partDataSelect, in2 := 14)
      Move(in := "Unit1.HmiInterface".PartData[14], out1 => "Unit1.EmData".PartData[14])
   END_RUNG
   RUNG wire#w1
      { S7_Templates := "SrcType := Int" } EQ_Contact(in1 := "Unit1.HmiInterface".partDataSelect, in2 := 15)
      Move(in := "Unit1.HmiInterface".PartData[15], out1 => "Unit1.EmData".PartData[15])
   END_RUNG
   RUNG wire#w1
      { S7_Templates := "SrcType := Int" } EQ_Contact(in1 := "Unit1.HmiInterface".partDataSelect, in2 := 16)
      Move(in := "Unit1.HmiInterface".PartData[16], out1 => "Unit1.EmData".PartData[16])
   END_RUNG
   RUNG wire#w1
      { S7_Templates := "SrcType := Int" } EQ_Contact(in1 := "Unit1.HmiInterface".partDataSelect, in2 := 17)
      Move(in := "Unit1.HmiInterface".PartData[17], out1 => "Unit1.EmData".PartData[17])
   END_RUNG
   RUNG wire#w1
      { S7_Templates := "SrcType := Int" } EQ_Contact(in1 := "Unit1.HmiInterface".partDataSelect, in2 := 18)
      Move(in := "Unit1.HmiInterface".PartData[18], out1 => "Unit1.EmData".PartData[18])
   END_RUNG
   // the same network as SCL:
   IF #instTonTimer[0].Q AND ("Unit1.HmiInterface".partDataSelect = 1) THEN
       "Unit1.EmData".PartData[1] := "Unit1.HmiInterface".PartData[1];
   END_IF;
   IF #instTonTimer[0].Q AND ("Unit1.HmiInterface".partDataSelect = 2) THEN
       "Unit1.EmData".PartData[2] := "Unit1.HmiInterface".PartData[2];
   END_IF;
   IF #instTonTimer[0].Q AND ("Unit1.HmiInterface".partDataSelect = 3) THEN
       "Unit1.EmData".PartData[3] := "Unit1.HmiInterface".PartData[3];
   END_IF;
   IF #instTonTimer[0].Q AND ("Unit1.HmiInterface".partDataSelect = 4) THEN
       "Unit1.EmData".PartData[4] := "Unit1.HmiInterface".PartData[4];
   END_IF;
   IF #instTonTimer[0].Q AND ("Unit1.HmiInterface".partDataSelect = 5) THEN
       "Unit1.EmData".PartData[5] := "Unit1.HmiInterface".PartData[5];
   END_IF;
   IF #instTonTimer[0].Q AND ("Unit1.HmiInterface".partDataSelect = 6) THEN
       "Unit1.EmData".PartData[6] := "Unit1.HmiInterface".PartData[6];
   END_IF;
   IF #instTonTimer[0].Q AND ("Unit1.HmiInterface".partDataSelect = 7) THEN
       "Unit1.EmData".PartData[7] := "Unit1.HmiInterface".PartData[7];
   END_IF;
   IF #instTonTimer[0].Q AND ("Unit1.HmiInterface".partDataSelect = 8) THEN
       "Unit1.EmData".PartData[8] := "Unit1.HmiInterface".PartData[8];
   END_IF;
   IF #instTonTimer[0].Q AND ("Unit1.HmiInterface".partDataSelect = 9) THEN
       "Unit1.EmData".PartData[9] := "Unit1.HmiInterface".PartData[9];
   END_IF;
   IF #instTonTimer[0].Q AND ("Unit1.HmiInterface".partDataSelect = 10) THEN
       "Unit1.EmData".PartData[10] := "Unit1.HmiInterface".PartData[10];
   END_IF;
   IF #instTonTimer[0].Q AND ("Unit1.HmiInterface".partDataSelect = 11) THEN
       "Unit1.EmData".PartData[11] := "Unit1.HmiInterface".PartData[11];
   END_IF;
   IF #instTonTimer[0].Q AND ("Unit1.HmiInterface".partDataSelect = 12) THEN
       "Unit1.EmData".PartData[12] := "Unit1.HmiInterface".PartData[12];
   END_IF;
   IF #instTonTimer[0].Q AND ("Unit1.HmiInterface".partDataSelect = 13) THEN
       "Unit1.EmData".PartData[13] := "Unit1.HmiInterface".PartData[13];
   END_IF;
   IF #instTonTimer[0].Q AND ("Unit1.HmiInterface".partDataSelect = 14) THEN
       "Unit1.EmData".PartData[14] := "Unit1.HmiInterface".PartData[14];
   END_IF;
   IF #instTonTimer[0].Q AND ("Unit1.HmiInterface".partDataSelect = 15) THEN
       "Unit1.EmData".PartData[15] := "Unit1.HmiInterface".PartData[15];
   END_IF;
   IF #instTonTimer[0].Q AND ("Unit1.HmiInterface".partDataSelect = 16) THEN
       "Unit1.EmData".PartData[16] := "Unit1.HmiInterface".PartData[16];
   END_IF;
   IF #instTonTimer[0].Q AND ("Unit1.HmiInterface".partDataSelect = 17) THEN
       "Unit1.EmData".PartData[17] := "Unit1.HmiInterface".PartData[17];
   END_IF;
   IF #instTonTimer[0].Q AND ("Unit1.HmiInterface".partDataSelect = 18) THEN
       "Unit1.EmData".PartData[18] := "Unit1.HmiInterface".PartData[18];
   END_IF;
END_REGION

REGION Network 82: Clear Command HMI -> Em Node
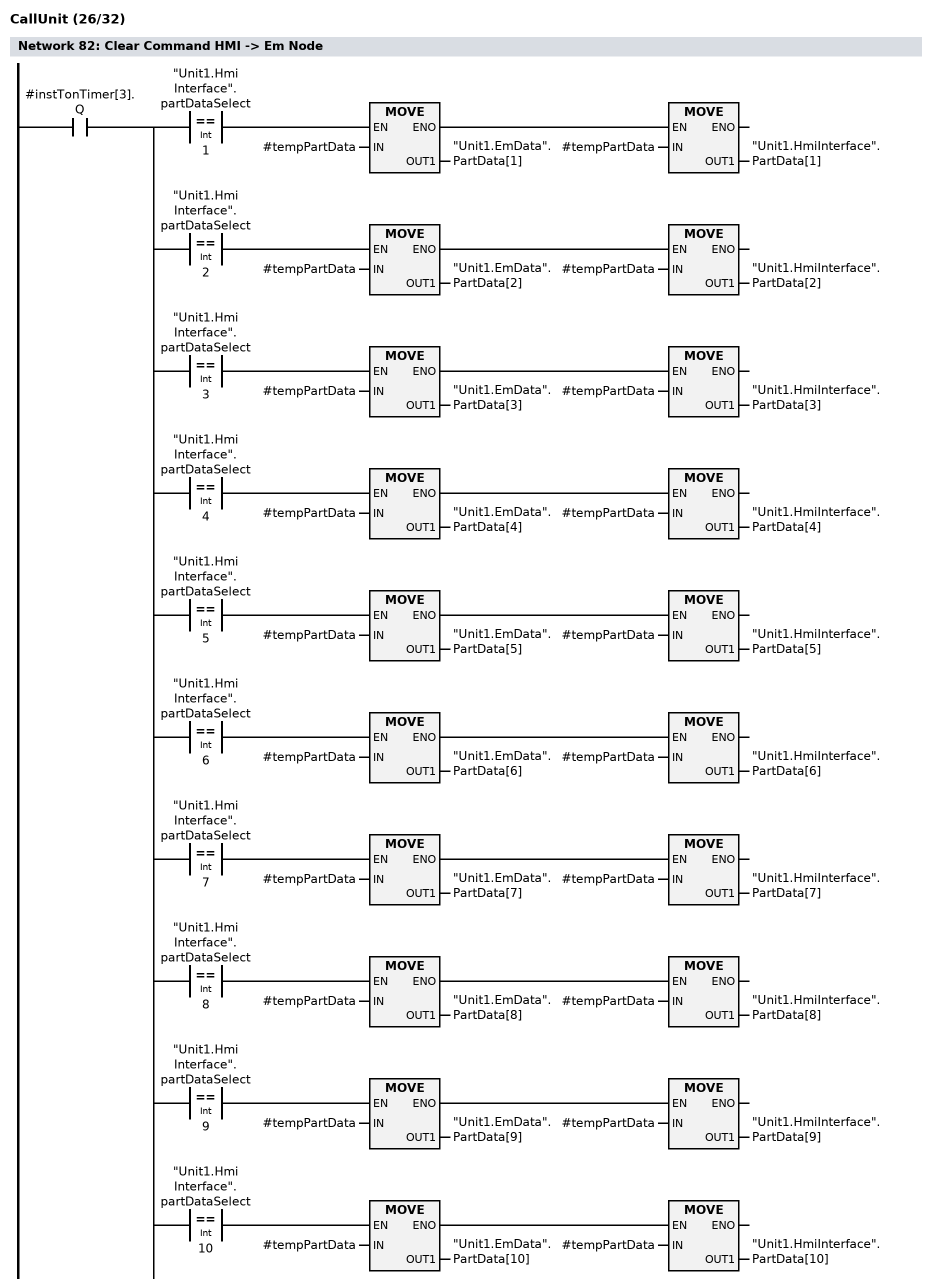
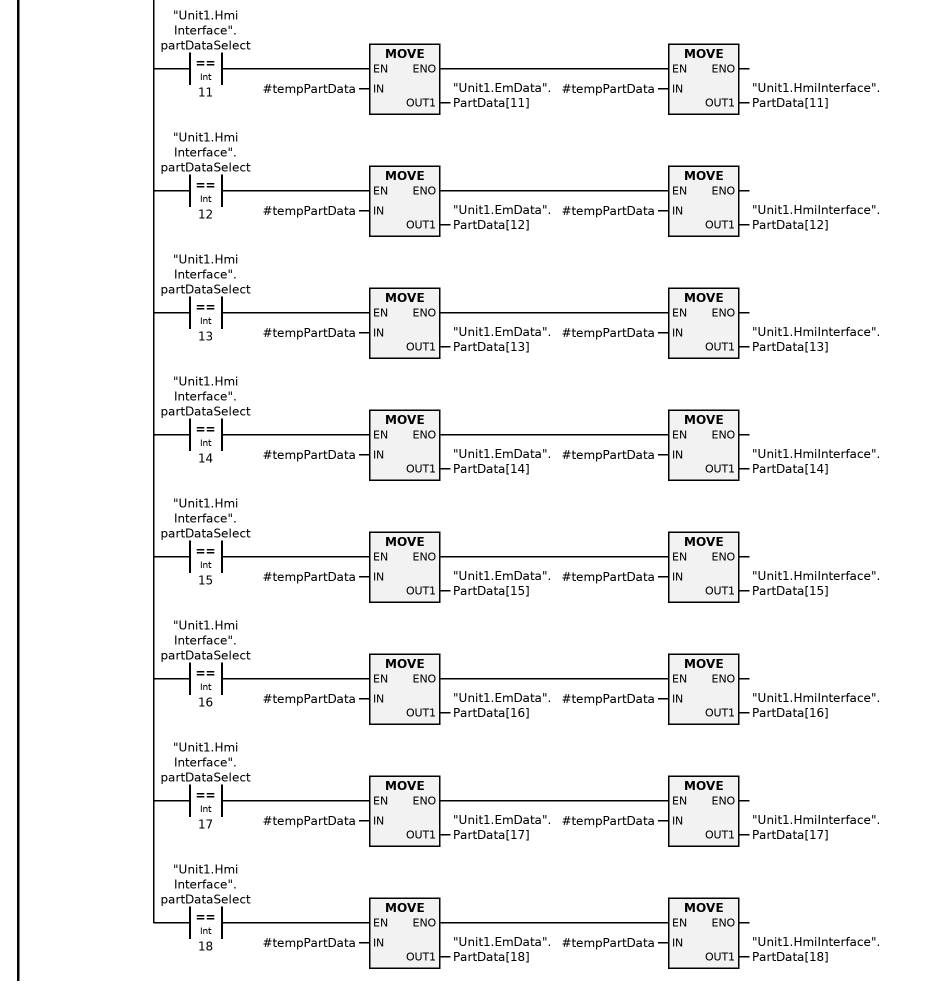
   RUNG wire#powerrail
      Contact( #instTonTimer[3].Q )
      wire#w1
      { S7_Templates := "SrcType := Int" } EQ_Contact(in1 := "Unit1.HmiInterface".partDataSelect, in2 := 1)
      Move(in := #tempPartData, out1 => "Unit1.EmData".PartData[1])
      Move(in := #tempPartData, out1 => "Unit1.HmiInterface".PartData[1])
   END_RUNG
   RUNG wire#w1
      { S7_Templates := "SrcType := Int" } EQ_Contact(in1 := "Unit1.HmiInterface".partDataSelect, in2 := 2)
      Move(in := #tempPartData, out1 => "Unit1.EmData".PartData[2])
      Move(in := #tempPartData, out1 => "Unit1.HmiInterface".PartData[2])
   END_RUNG
   RUNG wire#w1
      { S7_Templates := "SrcType := Int" } EQ_Contact(in1 := "Unit1.HmiInterface".partDataSelect, in2 := 3)
      Move(in := #tempPartData, out1 => "Unit1.EmData".PartData[3])
      Move(in := #tempPartData, out1 => "Unit1.HmiInterface".PartData[3])
   END_RUNG
   RUNG wire#w1
      { S7_Templates := "SrcType := Int" } EQ_Contact(in1 := "Unit1.HmiInterface".partDataSelect, in2 := 4)
      Move(in := #tempPartData, out1 => "Unit1.EmData".PartData[4])
      Move(in := #tempPartData, out1 => "Unit1.HmiInterface".PartData[4])
   END_RUNG
   RUNG wire#w1
      { S7_Templates := "SrcType := Int" } EQ_Contact(in1 := "Unit1.HmiInterface".partDataSelect, in2 := 5)
      Move(in := #tempPartData, out1 => "Unit1.EmData".PartData[5])
      Move(in := #tempPartData, out1 => "Unit1.HmiInterface".PartData[5])
   END_RUNG
   RUNG wire#w1
      { S7_Templates := "SrcType := Int" } EQ_Contact(in1 := "Unit1.HmiInterface".partDataSelect, in2 := 6)
      Move(in := #tempPartData, out1 => "Unit1.EmData".PartData[6])
      Move(in := #tempPartData, out1 => "Unit1.HmiInterface".PartData[6])
   END_RUNG
   RUNG wire#w1
      { S7_Templates := "SrcType := Int" } EQ_Contact(in1 := "Unit1.HmiInterface".partDataSelect, in2 := 7)
      Move(in := #tempPartData, out1 => "Unit1.EmData".PartData[7])
      Move(in := #tempPartData, out1 => "Unit1.HmiInterface".PartData[7])
   END_RUNG
   RUNG wire#w1
      { S7_Templates := "SrcType := Int" } EQ_Contact(in1 := "Unit1.HmiInterface".partDataSelect, in2 := 8)
      Move(in := #tempPartData, out1 => "Unit1.EmData".PartData[8])
      Move(in := #tempPartData, out1 => "Unit1.HmiInterface".PartData[8])
   END_RUNG
   RUNG wire#w1
      { S7_Templates := "SrcType := Int" } EQ_Contact(in1 := "Unit1.HmiInterface".partDataSelect, in2 := 9)
      Move(in := #tempPartData, out1 => "Unit1.EmData".PartData[9])
      Move(in := #tempPartData, out1 => "Unit1.HmiInterface".PartData[9])
   END_RUNG
   RUNG wire#w1
      { S7_Templates := "SrcType := Int" } EQ_Contact(in1 := "Unit1.HmiInterface".partDataSelect, in2 := 10)
      Move(in := #tempPartData, out1 => "Unit1.EmData".PartData[10])
      Move(in := #tempPartData, out1 => "Unit1.HmiInterface".PartData[10])
   END_RUNG
   RUNG wire#w1
      { S7_Templates := "SrcType := Int" } EQ_Contact(in1 := "Unit1.HmiInterface".partDataSelect, in2 := 11)
      Move(in := #tempPartData, out1 => "Unit1.EmData".PartData[11])
      Move(in := #tempPartData, out1 => "Unit1.HmiInterface".PartData[11])
   END_RUNG
   RUNG wire#w1
      { S7_Templates := "SrcType := Int" } EQ_Contact(in1 := "Unit1.HmiInterface".partDataSelect, in2 := 12)
      Move(in := #tempPartData, out1 => "Unit1.EmData".PartData[12])
      Move(in := #tempPartData, out1 => "Unit1.HmiInterface".PartData[12])
   END_RUNG
   RUNG wire#w1
      { S7_Templates := "SrcType := Int" } EQ_Contact(in1 := "Unit1.HmiInterface".partDataSelect, in2 := 13)
      Move(in := #tempPartData, out1 => "Unit1.EmData".PartData[13])
      Move(in := #tempPartData, out1 => "Unit1.HmiInterface".PartData[13])
   END_RUNG
   RUNG wire#w1
      { S7_Templates := "SrcType := Int" } EQ_Contact(in1 := "Unit1.HmiInterface".partDataSelect, in2 := 14)
      Move(in := #tempPartData, out1 => "Unit1.EmData".PartData[14])
      Move(in := #tempPartData, out1 => "Unit1.HmiInterface".PartData[14])
   END_RUNG
   RUNG wire#w1
      { S7_Templates := "SrcType := Int" } EQ_Contact(in1 := "Unit1.HmiInterface".partDataSelect, in2 := 15)
      Move(in := #tempPartData, out1 => "Unit1.EmData".PartData[15])
      Move(in := #tempPartData, out1 => "Unit1.HmiInterface".PartData[15])
   END_RUNG
   RUNG wire#w1
      { S7_Templates := "SrcType := Int" } EQ_Contact(in1 := "Unit1.HmiInterface".partDataSelect, in2 := 16)
      Move(in := #tempPartData, out1 => "Unit1.EmData".PartData[16])
      Move(in := #tempPartData, out1 => "Unit1.HmiInterface".PartData[16])
   END_RUNG
   RUNG wire#w1
      { S7_Templates := "SrcType := Int" } EQ_Contact(in1 := "Unit1.HmiInterface".partDataSelect, in2 := 17)
      Move(in := #tempPartData, out1 => "Unit1.EmData".PartData[17])
      Move(in := #tempPartData, out1 => "Unit1.HmiInterface".PartData[17])
   END_RUNG
   RUNG wire#w1
      { S7_Templates := "SrcType := Int" } EQ_Contact(in1 := "Unit1.HmiInterface".partDataSelect, in2 := 18)
      Move(in := #tempPartData, out1 => "Unit1.EmData".PartData[18])
      Move(in := #tempPartData, out1 => "Unit1.HmiInterface".PartData[18])
   END_RUNG
   // the same network as SCL:
   IF #instTonTimer[3].Q AND ("Unit1.HmiInterface".partDataSelect = 1) THEN
       "Unit1.EmData".PartData[1] := #tempPartData;
       "Unit1.HmiInterface".PartData[1] := #tempPartData;
   END_IF;
   IF #instTonTimer[3].Q AND ("Unit1.HmiInterface".partDataSelect = 2) THEN
       "Unit1.EmData".PartData[2] := #tempPartData;
       "Unit1.HmiInterface".PartData[2] := #tempPartData;
   END_IF;
   IF #instTonTimer[3].Q AND ("Unit1.HmiInterface".partDataSelect = 3) THEN
       "Unit1.EmData".PartData[3] := #tempPartData;
       "Unit1.HmiInterface".PartData[3] := #tempPartData;
   END_IF;
   IF #instTonTimer[3].Q AND ("Unit1.HmiInterface".partDataSelect = 4) THEN
       "Unit1.EmData".PartData[4] := #tempPartData;
       "Unit1.HmiInterface".PartData[4] := #tempPartData;
   END_IF;
   IF #instTonTimer[3].Q AND ("Unit1.HmiInterface".partDataSelect = 5) THEN
       "Unit1.EmData".PartData[5] := #tempPartData;
       "Unit1.HmiInterface".PartData[5] := #tempPartData;
   END_IF;
   IF #instTonTimer[3].Q AND ("Unit1.HmiInterface".partDataSelect = 6) THEN
       "Unit1.EmData".PartData[6] := #tempPartData;
       "Unit1.HmiInterface".PartData[6] := #tempPartData;
   END_IF;
   IF #instTonTimer[3].Q AND ("Unit1.HmiInterface".partDataSelect = 7) THEN
       "Unit1.EmData".PartData[7] := #tempPartData;
       "Unit1.HmiInterface".PartData[7] := #tempPartData;
   END_IF;
   IF #instTonTimer[3].Q AND ("Unit1.HmiInterface".partDataSelect = 8) THEN
       "Unit1.EmData".PartData[8] := #tempPartData;
       "Unit1.HmiInterface".PartData[8] := #tempPartData;
   END_IF;
   IF #instTonTimer[3].Q AND ("Unit1.HmiInterface".partDataSelect = 9) THEN
       "Unit1.EmData".PartData[9] := #tempPartData;
       "Unit1.HmiInterface".PartData[9] := #tempPartData;
   END_IF;
   IF #instTonTimer[3].Q AND ("Unit1.HmiInterface".partDataSelect = 10) THEN
       "Unit1.EmData".PartData[10] := #tempPartData;
       "Unit1.HmiInterface".PartData[10] := #tempPartData;
   END_IF;
   IF #instTonTimer[3].Q AND ("Unit1.HmiInterface".partDataSelect = 11) THEN
       "Unit1.EmData".PartData[11] := #tempPartData;
       "Unit1.HmiInterface".PartData[11] := #tempPartData;
   END_IF;
   IF #instTonTimer[3].Q AND ("Unit1.HmiInterface".partDataSelect = 12) THEN
       "Unit1.EmData".PartData[12] := #tempPartData;
       "Unit1.HmiInterface".PartData[12] := #tempPartData;
   END_IF;
   IF #instTonTimer[3].Q AND ("Unit1.HmiInterface".partDataSelect = 13) THEN
       "Unit1.EmData".PartData[13] := #tempPartData;
       "Unit1.HmiInterface".PartData[13] := #tempPartData;
   END_IF;
   IF #instTonTimer[3].Q AND ("Unit1.HmiInterface".partDataSelect = 14) THEN
       "Unit1.EmData".PartData[14] := #tempPartData;
       "Unit1.HmiInterface".PartData[14] := #tempPartData;
   END_IF;
   IF #instTonTimer[3].Q AND ("Unit1.HmiInterface".partDataSelect = 15) THEN
       "Unit1.EmData".PartData[15] := #tempPartData;
       "Unit1.HmiInterface".PartData[15] := #tempPartData;
   END_IF;
   IF #instTonTimer[3].Q AND ("Unit1.HmiInterface".partDataSelect = 16) THEN
       "Unit1.EmData".PartData[16] := #tempPartData;
       "Unit1.HmiInterface".PartData[16] := #tempPartData;
   END_IF;
   IF #instTonTimer[3].Q AND ("Unit1.HmiInterface".partDataSelect = 17) THEN
       "Unit1.EmData".PartData[17] := #tempPartData;
       "Unit1.HmiInterface".PartData[17] := #tempPartData;
   END_IF;
   IF #instTonTimer[3].Q AND ("Unit1.HmiInterface".partDataSelect = 18) THEN
       "Unit1.EmData".PartData[18] := #tempPartData;
       "Unit1.HmiInterface".PartData[18] := #tempPartData;
   END_IF;
END_REGION

REGION Network 83: All Clear Command HMI -> Em Node
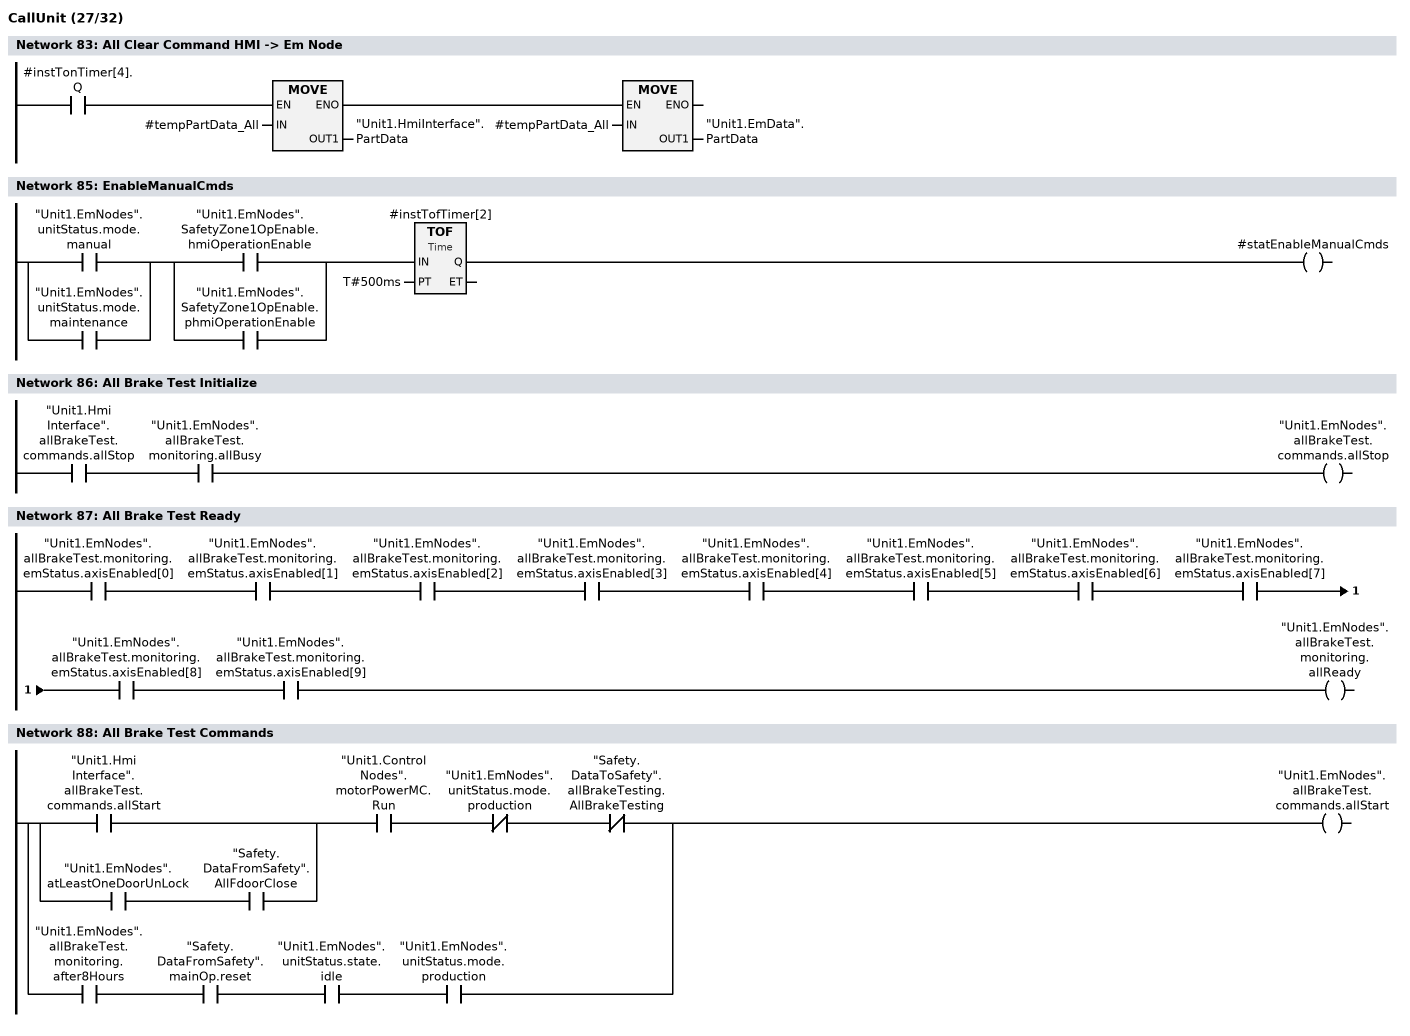
   RUNG wire#powerrail
      Contact( #instTonTimer[4].Q )
      Move(in := #tempPartData_All, out1 => "Unit1.HmiInterface".PartData)
      Move(in := #tempPartData_All, out1 => "Unit1.EmData".PartData)
   END_RUNG
   // the same network as SCL:
   IF #instTonTimer[4].Q THEN
       "Unit1.HmiInterface".PartData := #tempPartData_All;
       "Unit1.EmData".PartData := #tempPartData_All;
   END_IF;
END_REGION

REGION Network 84: ******************** Brake Test ********************
END_REGION

REGION Network 85: EnableManualCmds
   RUNG wire#powerrail
      Contact( "Unit1.EmNodes".unitStatus.mode.manual )
      wire#w1
      Contact( "Unit1.EmNodes".SafetyZone1OpEnable.hmiOperationEnable )
      wire#w2
      { S7_Templates := "time_type := Time" } #instTofTimer[2].TOF(pt := T#500ms, et =>)
      Coil( #statEnableManualCmds )
   END_RUNG
   RUNG wire#powerrail
      Contact( "Unit1.EmNodes".unitStatus.mode.maintenance )
   END_RUNG wire#w1
   RUNG wire#w1
      Contact( "Unit1.EmNodes".SafetyZone1OpEnable.phmiOperationEnable )
   END_RUNG wire#w2
   // the same network as SCL:
   #instTofTimer[2].TOF(IN := ("Unit1.EmNodes".unitStatus.mode.manual OR "Unit1.EmNodes".unitStatus.mode.maintenance) AND ("Unit1.EmNodes".SafetyZone1OpEnable.hmiOperationEnable OR "Unit1.EmNodes".SafetyZone1OpEnable.phmiOperationEnable),
                        PT := T#500ms);
   #statEnableManualCmds := #instTofTimer[2].Q;
END_REGION

REGION Network 86: All Brake Test Initialize
   RUNG wire#powerrail
      Contact( "Unit1.HmiInterface".allBrakeTest.commands.allStop )
      Contact( "Unit1.EmNodes".allBrakeTest.monitoring.allBusy )
      Coil( "Unit1.EmNodes".allBrakeTest.commands.allStop )
   END_RUNG
   // the same network as SCL:
   "Unit1.EmNodes".allBrakeTest.commands.allStop := "Unit1.HmiInterface".allBrakeTest.commands.allStop AND "Unit1.EmNodes".allBrakeTest.monitoring.allBusy;
END_REGION

REGION Network 87: All Brake Test Ready
   RUNG wire#powerrail
      Contact( "Unit1.EmNodes".allBrakeTest.monitoring.emStatus.axisEnabled[0] )
      Contact( "Unit1.EmNodes".allBrakeTest.monitoring.emStatus.axisEnabled[1] )
      Contact( "Unit1.EmNodes".allBrakeTest.monitoring.emStatus.axisEnabled[2] )
      Contact( "Unit1.EmNodes".allBrakeTest.monitoring.emStatus.axisEnabled[3] )
      Contact( "Unit1.EmNodes".allBrakeTest.monitoring.emStatus.axisEnabled[4] )
      Contact( "Unit1.EmNodes".allBrakeTest.monitoring.emStatus.axisEnabled[5] )
      Contact( "Unit1.EmNodes".allBrakeTest.monitoring.emStatus.axisEnabled[6] )
      Contact( "Unit1.EmNodes".allBrakeTest.monitoring.emStatus.axisEnabled[7] )
      Contact( "Unit1.EmNodes".allBrakeTest.monitoring.emStatus.axisEnabled[8] )
      Contact( "Unit1.EmNodes".allBrakeTest.monitoring.emStatus.axisEnabled[9] )
      Coil( "Unit1.EmNodes".allBrakeTest.monitoring.allReady )
   END_RUNG
   // the same network as SCL:
   "Unit1.EmNodes".allBrakeTest.monitoring.allReady := "Unit1.EmNodes".allBrakeTest.monitoring.emStatus.axisEnabled[0] AND "Unit1.EmNodes".allBrakeTest.monitoring.emStatus.axisEnabled[1] AND "Unit1.EmNodes".allBrakeTest.monitoring.emStatus.axisEnabled[2] AND "Unit1.EmNodes".allBrakeTest.monitoring.emStatus.axisEnabled[3] AND "Unit1.EmNodes".allBrakeTest.monitoring.emStatus.axisEnabled[4] AND "Unit1.EmNodes".allBrakeTest.monitoring.emStatus.axisEnabled[5] AND "Unit1.EmNodes".allBrakeTest.monitoring.emStatus.axisEnabled[6] AND "Unit1.EmNodes".allBrakeTest.monitoring.emStatus.axisEnabled[7] AND "Unit1.EmNodes".allBrakeTest.monitoring.emStatus.axisEnabled[8] AND "Unit1.EmNodes".allBrakeTest.monitoring.emStatus.axisEnabled[9];
END_REGION

REGION Network 88: All Brake Test Commands
   RUNG wire#powerrail
      Contact( "Unit1.HmiInterface".allBrakeTest.commands.allStart )
      wire#w1
      Contact( "Unit1.ControlNodes".motorPowerMC.Run )
      I_Contact( "Unit1.EmNodes".unitStatus.mode.production )
      I_Contact( "Safety.DataToSafety".allBrakeTesting.AllBrakeTesting )
      wire#w2
      Coil( "Unit1.EmNodes".allBrakeTest.commands.allStart )
   END_RUNG
   RUNG wire#powerrail
      Contact( "Unit1.EmNodes".atLeastOneDoorUnLock )
      Contact( "Safety.DataFromSafety".AllFdoorClose )
   END_RUNG wire#w1
   RUNG wire#powerrail
      Contact( "Unit1.EmNodes".allBrakeTest.monitoring.after8Hours )
      Contact( "Safety.DataFromSafety".mainOp.reset )
      Contact( "Unit1.EmNodes".unitStatus.state.idle )
      Contact( "Unit1.EmNodes".unitStatus.mode.production )
   END_RUNG wire#w2
   // the same network as SCL:
   "Unit1.EmNodes".allBrakeTest.commands.allStart := (("Unit1.HmiInterface".allBrakeTest.commands.allStart OR ("Unit1.EmNodes".atLeastOneDoorUnLock AND "Safety.DataFromSafety".AllFdoorClose)) AND "Unit1.ControlNodes".motorPowerMC.Run AND NOT "Unit1.EmNodes".unitStatus.mode.production AND NOT "Safety.DataToSafety".allBrakeTesting.AllBrakeTesting) OR ("Unit1.EmNodes".allBrakeTest.monitoring.after8Hours AND "Safety.DataFromSafety".mainOp.reset AND "Unit1.EmNodes".unitStatus.state.idle AND "Unit1.EmNodes".unitStatus.mode.production);
END_REGION

REGION Network 89: Em Brake Test Status Summary
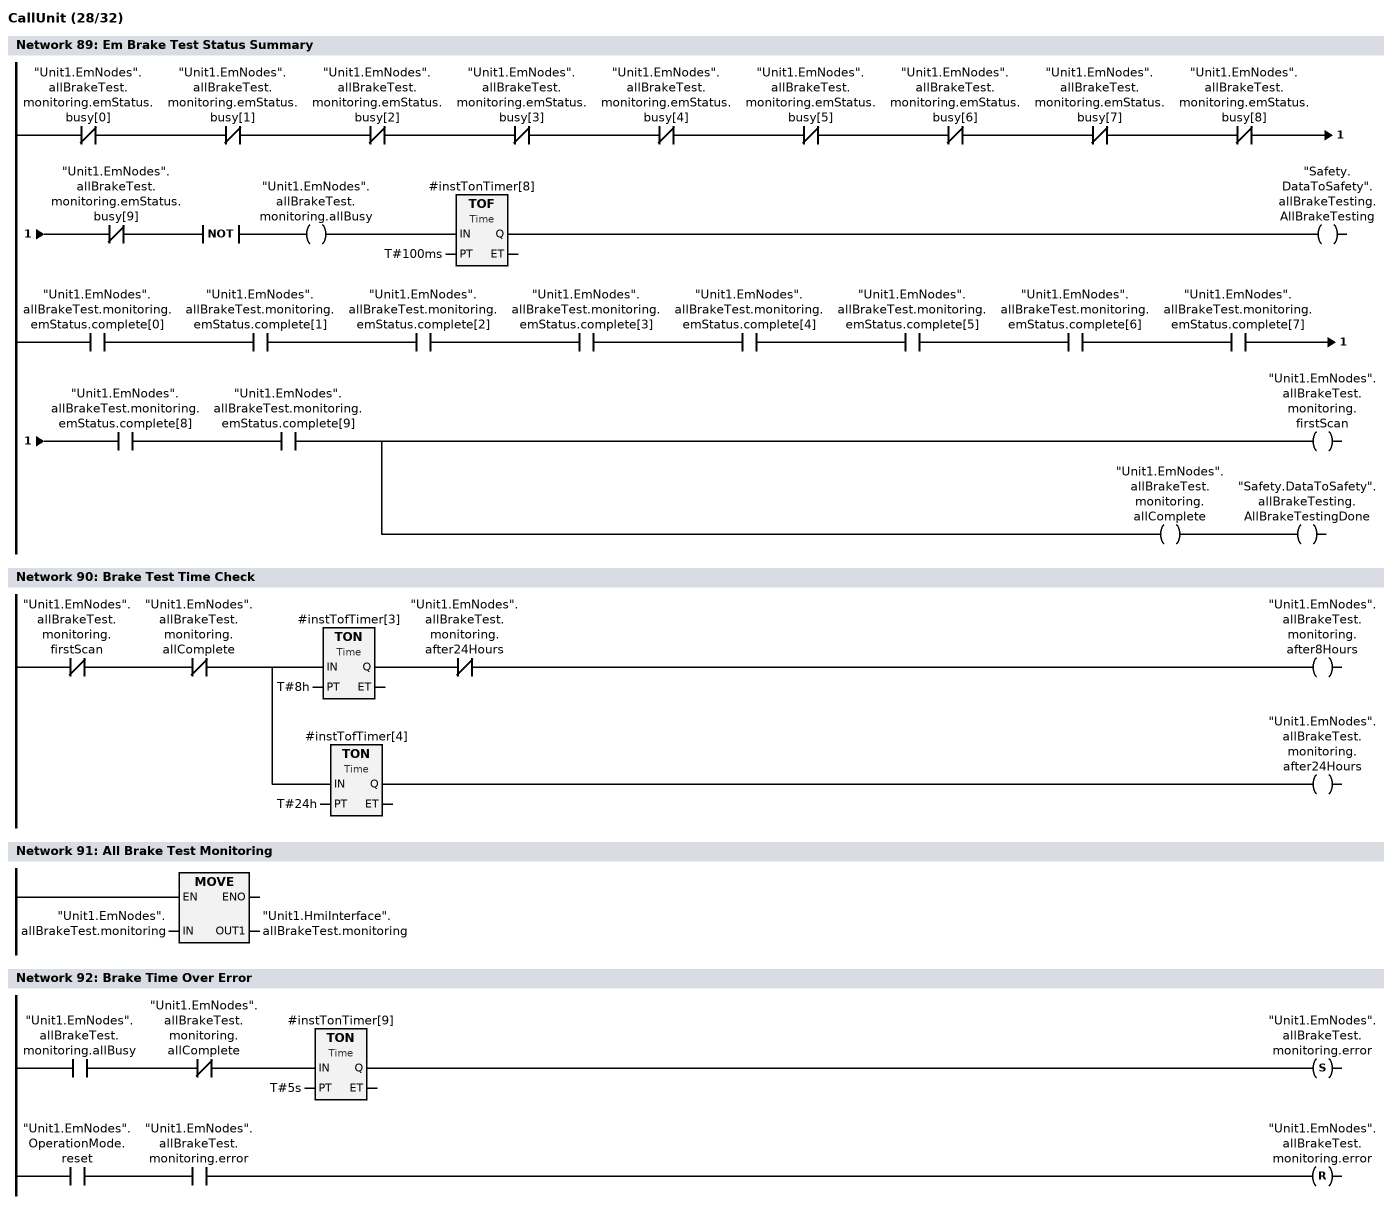
   RUNG wire#powerrail
      I_Contact( "Unit1.EmNodes".allBrakeTest.monitoring.emStatus.busy[0] )
      I_Contact( "Unit1.EmNodes".allBrakeTest.monitoring.emStatus.busy[1] )
      I_Contact( "Unit1.EmNodes".allBrakeTest.monitoring.emStatus.busy[2] )
      I_Contact( "Unit1.EmNodes".allBrakeTest.monitoring.emStatus.busy[3] )
      I_Contact( "Unit1.EmNodes".allBrakeTest.monitoring.emStatus.busy[4] )
      I_Contact( "Unit1.EmNodes".allBrakeTest.monitoring.emStatus.busy[5] )
      I_Contact( "Unit1.EmNodes".allBrakeTest.monitoring.emStatus.busy[6] )
      I_Contact( "Unit1.EmNodes".allBrakeTest.monitoring.emStatus.busy[7] )
      I_Contact( "Unit1.EmNodes".allBrakeTest.monitoring.emStatus.busy[8] )
      I_Contact( "Unit1.EmNodes".allBrakeTest.monitoring.emStatus.busy[9] )
      Not()
      Coil( "Unit1.EmNodes".allBrakeTest.monitoring.allBusy )
      { S7_Templates := "time_type := Time" } #instTonTimer[8].TOF(pt := T#100ms, et =>)
      Coil( "Safety.DataToSafety".allBrakeTesting.AllBrakeTesting )
   END_RUNG
   RUNG wire#powerrail
      Contact( "Unit1.EmNodes".allBrakeTest.monitoring.emStatus.complete[0] )
      Contact( "Unit1.EmNodes".allBrakeTest.monitoring.emStatus.complete[1] )
      Contact( "Unit1.EmNodes".allBrakeTest.monitoring.emStatus.complete[2] )
      Contact( "Unit1.EmNodes".allBrakeTest.monitoring.emStatus.complete[3] )
      Contact( "Unit1.EmNodes".allBrakeTest.monitoring.emStatus.complete[4] )
      Contact( "Unit1.EmNodes".allBrakeTest.monitoring.emStatus.complete[5] )
      Contact( "Unit1.EmNodes".allBrakeTest.monitoring.emStatus.complete[6] )
      Contact( "Unit1.EmNodes".allBrakeTest.monitoring.emStatus.complete[7] )
      Contact( "Unit1.EmNodes".allBrakeTest.monitoring.emStatus.complete[8] )
      Contact( "Unit1.EmNodes".allBrakeTest.monitoring.emStatus.complete[9] )
      wire#w1
      Coil( "Unit1.EmNodes".allBrakeTest.monitoring.firstScan )
   END_RUNG
   RUNG wire#w1
      Coil( "Unit1.EmNodes".allBrakeTest.monitoring.allComplete )
      Coil( "Safety.DataToSafety".allBrakeTesting.AllBrakeTestingDone )
   END_RUNG
   // the same network as SCL:
   "Unit1.EmNodes".allBrakeTest.monitoring.allBusy := NOT (NOT "Unit1.EmNodes".allBrakeTest.monitoring.emStatus.busy[0] AND NOT "Unit1.EmNodes".allBrakeTest.monitoring.emStatus.busy[1] AND NOT "Unit1.EmNodes".allBrakeTest.monitoring.emStatus.busy[2] AND NOT "Unit1.EmNodes".allBrakeTest.monitoring.emStatus.busy[3] AND NOT "Unit1.EmNodes".allBrakeTest.monitoring.emStatus.busy[4] AND NOT "Unit1.EmNodes".allBrakeTest.monitoring.emStatus.busy[5] AND NOT "Unit1.EmNodes".allBrakeTest.monitoring.emStatus.busy[6] AND NOT "Unit1.EmNodes".allBrakeTest.monitoring.emStatus.busy[7] AND NOT "Unit1.EmNodes".allBrakeTest.monitoring.emStatus.busy[8] AND NOT "Unit1.EmNodes".allBrakeTest.monitoring.emStatus.busy[9]);
   #instTonTimer[8].TOF(IN := "Unit1.EmNodes".allBrakeTest.monitoring.allBusy, PT := T#100ms);
   "Safety.DataToSafety".allBrakeTesting.AllBrakeTesting := #instTonTimer[8].Q;
   "Unit1.EmNodes".allBrakeTest.monitoring.firstScan := "Unit1.EmNodes".allBrakeTest.monitoring.emStatus.complete[0] AND "Unit1.EmNodes".allBrakeTest.monitoring.emStatus.complete[1] AND "Unit1.EmNodes".allBrakeTest.monitoring.emStatus.complete[2] AND "Unit1.EmNodes".allBrakeTest.monitoring.emStatus.complete[3] AND "Unit1.EmNodes".allBrakeTest.monitoring.emStatus.complete[4] AND "Unit1.EmNodes".allBrakeTest.monitoring.emStatus.complete[5] AND "Unit1.EmNodes".allBrakeTest.monitoring.emStatus.complete[6] AND "Unit1.EmNodes".allBrakeTest.monitoring.emStatus.complete[7] AND "Unit1.EmNodes".allBrakeTest.monitoring.emStatus.complete[8] AND "Unit1.EmNodes".allBrakeTest.monitoring.emStatus.complete[9];
   "Unit1.EmNodes".allBrakeTest.monitoring.allComplete := "Unit1.EmNodes".allBrakeTest.monitoring.firstScan;
   "Safety.DataToSafety".allBrakeTesting.AllBrakeTestingDone := "Unit1.EmNodes".allBrakeTest.monitoring.firstScan;
END_REGION

REGION Network 90: Brake Test Time Check
   RUNG wire#powerrail
      I_Contact( "Unit1.EmNodes".allBrakeTest.monitoring.firstScan )
      I_Contact( "Unit1.EmNodes".allBrakeTest.monitoring.allComplete )
      wire#w1
      { S7_Templates := "time_type := Time" } #instTofTimer[3].TON(pt := T#8h, et =>)
      I_Contact( "Unit1.EmNodes".allBrakeTest.monitoring.after24Hours )
      Coil( "Unit1.EmNodes".allBrakeTest.monitoring.after8Hours )
   END_RUNG
   RUNG wire#w1
      { S7_Templates := "time_type := Time" } #instTofTimer[4].TON(pt := T#24h, et =>)
      Coil( "Unit1.EmNodes".allBrakeTest.monitoring.after24Hours )
   END_RUNG
   // the same network as SCL:
   #_w1 := NOT "Unit1.EmNodes".allBrakeTest.monitoring.firstScan AND NOT "Unit1.EmNodes".allBrakeTest.monitoring.allComplete;
   #instTofTimer[3].TON(IN := #_w1, PT := T#8h);
   "Unit1.EmNodes".allBrakeTest.monitoring.after8Hours := #instTofTimer[3].Q AND NOT "Unit1.EmNodes".allBrakeTest.monitoring.after24Hours;
   #instTofTimer[4].TON(IN := #_w1, PT := T#24h);
   "Unit1.EmNodes".allBrakeTest.monitoring.after24Hours := #instTofTimer[4].Q;
END_REGION

REGION Network 91: All Brake Test Monitoring
   RUNG wire#powerrail
      Move(in := "Unit1.EmNodes".allBrakeTest.monitoring, out1 => "Unit1.HmiInterface".allBrakeTest.monitoring)
   END_RUNG
   // the same network as SCL:
   "Unit1.HmiInterface".allBrakeTest.monitoring := "Unit1.EmNodes".allBrakeTest.monitoring;
END_REGION

REGION Network 92: Brake Time Over Error
   RUNG wire#powerrail
      Contact( "Unit1.EmNodes".allBrakeTest.monitoring.allBusy )
      I_Contact( "Unit1.EmNodes".allBrakeTest.monitoring.allComplete )
      { S7_Templates := "time_type := Time" } #instTonTimer[9].TON(pt := T#5s, et =>)
      S_Coil( "Unit1.EmNodes".allBrakeTest.monitoring.error )
   END_RUNG
   RUNG wire#powerrail
      Contact( "Unit1.EmNodes".OperationMode.reset )
      Contact( "Unit1.EmNodes".allBrakeTest.monitoring.error )
      R_Coil( "Unit1.EmNodes".allBrakeTest.monitoring.error )
   END_RUNG
   // the same network as SCL:
   #instTonTimer[9].TON(IN := "Unit1.EmNodes".allBrakeTest.monitoring.allBusy AND NOT "Unit1.EmNodes".allBrakeTest.monitoring.allComplete,
                        PT := T#5s);
   IF #instTonTimer[9].Q THEN "Unit1.EmNodes".allBrakeTest.monitoring.error := TRUE; END_IF;
   IF "Unit1.EmNodes".OperationMode.reset AND "Unit1.EmNodes".allBrakeTest.monitoring.error THEN
       "Unit1.EmNodes".allBrakeTest.monitoring.error := FALSE;
   END_IF;
END_REGION

REGION Network 93: ******************** FFU LIU117 (MCU) ********************
END_REGION

REGION Network 94: CM LER_FFU_LIU117 Command
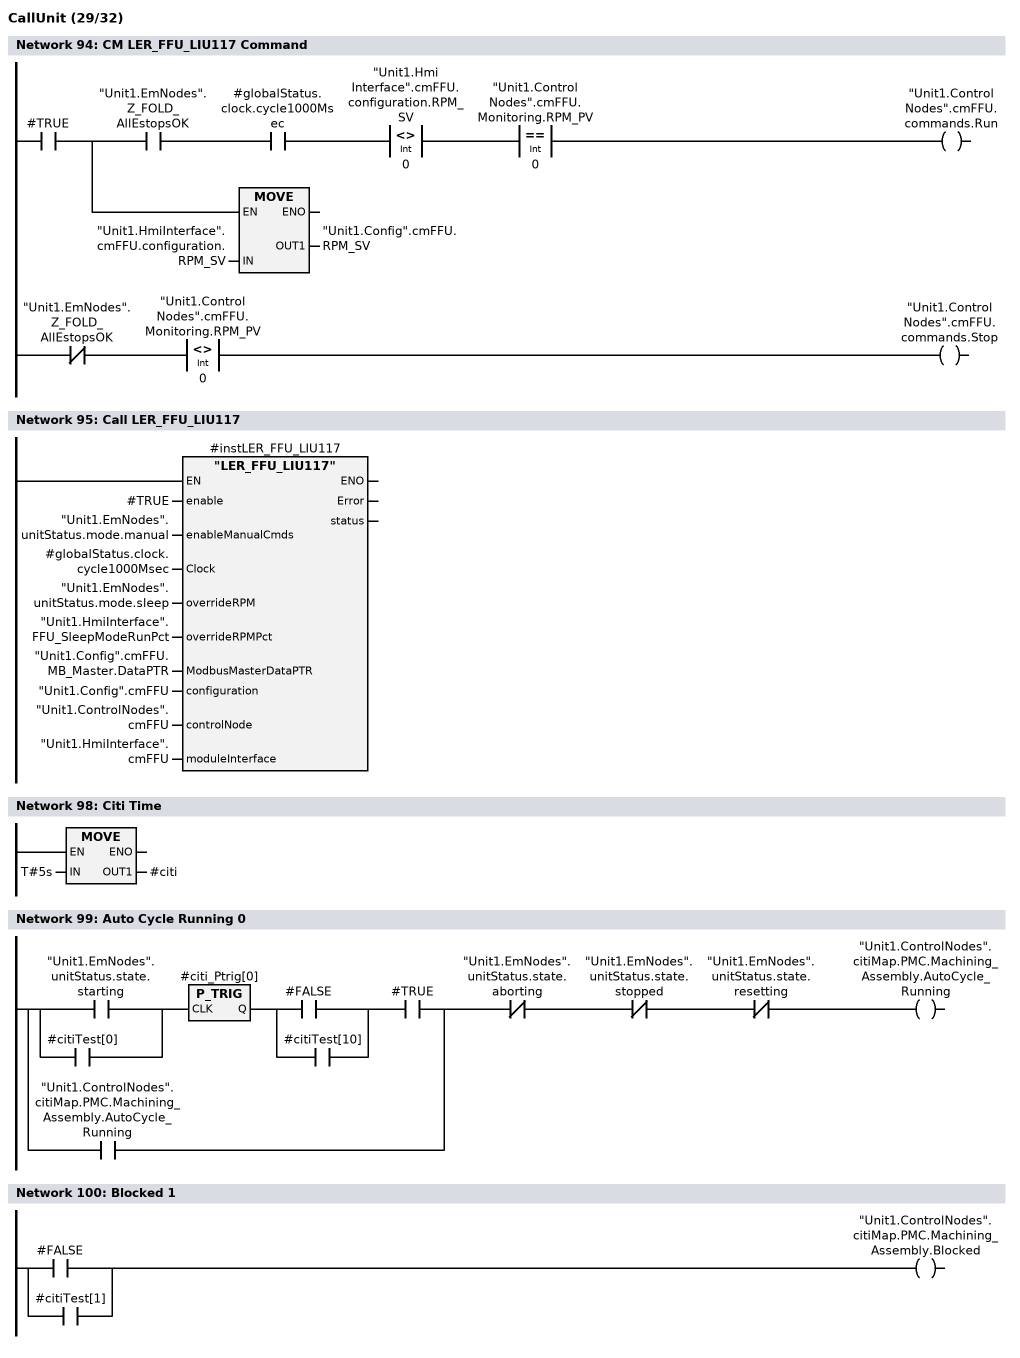
   RUNG wire#powerrail
      Contact( #TRUE )
      wire#w1
      Contact( "Unit1.EmNodes".Z_FOLD_AllEstopsOK )
      Contact( #globalStatus.clock.cycle1000Msec )
      { S7_Templates := "SrcType := Int" } NE_Contact(in1 := "Unit1.HmiInterface".cmFFU.configuration.RPM_SV, in2 := 0)
      { S7_Templates := "SrcType := Int" } EQ_Contact(in1 := "Unit1.ControlNodes".cmFFU.Monitoring.RPM_PV, in2 := 0)
      Coil( "Unit1.ControlNodes".cmFFU.commands.Run )
   END_RUNG
   RUNG wire#w1
      Move(in := "Unit1.HmiInterface".cmFFU.configuration.RPM_SV, out1 => "Unit1.Config".cmFFU.RPM_SV)
   END_RUNG
   RUNG wire#powerrail
      I_Contact( "Unit1.EmNodes".Z_FOLD_AllEstopsOK )
      { S7_Templates := "SrcType := Int" } NE_Contact(in1 := "Unit1.ControlNodes".cmFFU.Monitoring.RPM_PV, in2 := 0)
      Coil( "Unit1.ControlNodes".cmFFU.commands.Stop )
   END_RUNG
   // the same network as SCL:
   "Unit1.ControlNodes".cmFFU.commands.Run := #TRUE AND "Unit1.EmNodes".Z_FOLD_AllEstopsOK AND #globalStatus.clock.cycle1000Msec AND ("Unit1.HmiInterface".cmFFU.configuration.RPM_SV <> 0) AND ("Unit1.ControlNodes".cmFFU.Monitoring.RPM_PV = 0);
   IF #TRUE THEN "Unit1.Config".cmFFU.RPM_SV := "Unit1.HmiInterface".cmFFU.configuration.RPM_SV; END_IF;
   "Unit1.ControlNodes".cmFFU.commands.Stop := NOT "Unit1.EmNodes".Z_FOLD_AllEstopsOK AND ("Unit1.ControlNodes".cmFFU.Monitoring.RPM_PV <> 0);
END_REGION

REGION Network 95: Call LER_FFU_LIU117
   RUNG wire#powerrail
      #instLER_FFU_LIU117(enable := #TRUE, enableManualCmds := "Unit1.EmNodes".unitStatus.mode.manual, Clock := #globalStatus.clock.cycle1000Msec, overrideRPM := "Unit1.EmNodes".unitStatus.mode.sleep, overrideRPMPct := "Unit1.HmiInterface".FFU_SleepModeRunPct, ModbusMasterDataPTR := "Unit1.Config".cmFFU.MB_Master.DataPTR, configuration := "Unit1.Config".cmFFU, controlNode := "Unit1.ControlNodes".cmFFU, moduleInterface := "Unit1.HmiInterface".cmFFU, Error =>, status =>)
   END_RUNG
   // the same network as SCL:
   #instLER_FFU_LIU117(enable := #TRUE,   // "LER_FFU_LIU117"
                       enableManualCmds := "Unit1.EmNodes".unitStatus.mode.manual,
                       Clock := #globalStatus.clock.cycle1000Msec,
                       overrideRPM := "Unit1.EmNodes".unitStatus.mode.sleep,
                       overrideRPMPct := "Unit1.HmiInterface".FFU_SleepModeRunPct,
                       ModbusMasterDataPTR := "Unit1.Config".cmFFU.MB_Master.DataPTR,
                       configuration := "Unit1.Config".cmFFU,
                       controlNode := "Unit1.ControlNodes".cmFFU,
                       moduleInterface := "Unit1.HmiInterface".cmFFU);
END_REGION

REGION Network 97: ******************** CITI ********************
END_REGION

REGION Network 98: Citi Time
   RUNG wire#powerrail
      Move(in := T#5s, out1 => #citi)
   END_RUNG
   // the same network as SCL:
   #citi := T#5s;
END_REGION

REGION Network 99: Auto Cycle Running 0
   RUNG wire#powerrail
      Contact( "Unit1.EmNodes".unitStatus.state.starting )
      wire#w1
      P_Trig( #citi_Ptrig[0] )
      wire#w2
      Contact( #FALSE )
      wire#w3
      Contact( #TRUE )
      wire#w4
      I_Contact( "Unit1.EmNodes".unitStatus.state.aborting )
      I_Contact( "Unit1.EmNodes".unitStatus.state.stopped )
      I_Contact( "Unit1.EmNodes".unitStatus.state.resetting )
      Coil( "Unit1.ControlNodes".citiMap.PMC.Machining_Assembly.AutoCycle_Running )
   END_RUNG
   RUNG wire#powerrail
      Contact( #citiTest[0] )
   END_RUNG wire#w1
   RUNG wire#w2
      Contact( #citiTest[10] )
   END_RUNG wire#w3
   RUNG wire#powerrail
      Contact( "Unit1.ControlNodes".citiMap.PMC.Machining_Assembly.AutoCycle_Running )
   END_RUNG wire#w4
   // the same network as SCL:
   #_w1 := "Unit1.EmNodes".unitStatus.state.starting OR #citiTest[0];
   #_w2 := #_w1 AND NOT #citi_Ptrig[0];   // rising edge
   #citi_Ptrig[0] := #_w1;
   "Unit1.ControlNodes".citiMap.PMC.Machining_Assembly.AutoCycle_Running := ((#_w2 AND (#FALSE OR #citiTest[10]) AND #TRUE) OR "Unit1.ControlNodes".citiMap.PMC.Machining_Assembly.AutoCycle_Running) AND NOT "Unit1.EmNodes".unitStatus.state.aborting AND NOT "Unit1.EmNodes".unitStatus.state.stopped AND NOT "Unit1.EmNodes".unitStatus.state.resetting;
END_REGION

REGION Network 100: Blocked 1
   RUNG wire#powerrail
      Contact( #FALSE )
      wire#w1
      Coil( "Unit1.ControlNodes".citiMap.PMC.Machining_Assembly.Blocked )
   END_RUNG
   RUNG wire#powerrail
      Contact( #citiTest[1] )
   END_RUNG wire#w1
   // the same network as SCL:
   "Unit1.ControlNodes".citiMap.PMC.Machining_Assembly.Blocked := #FALSE OR #citiTest[1];
END_REGION

REGION Network 101: Starved 2
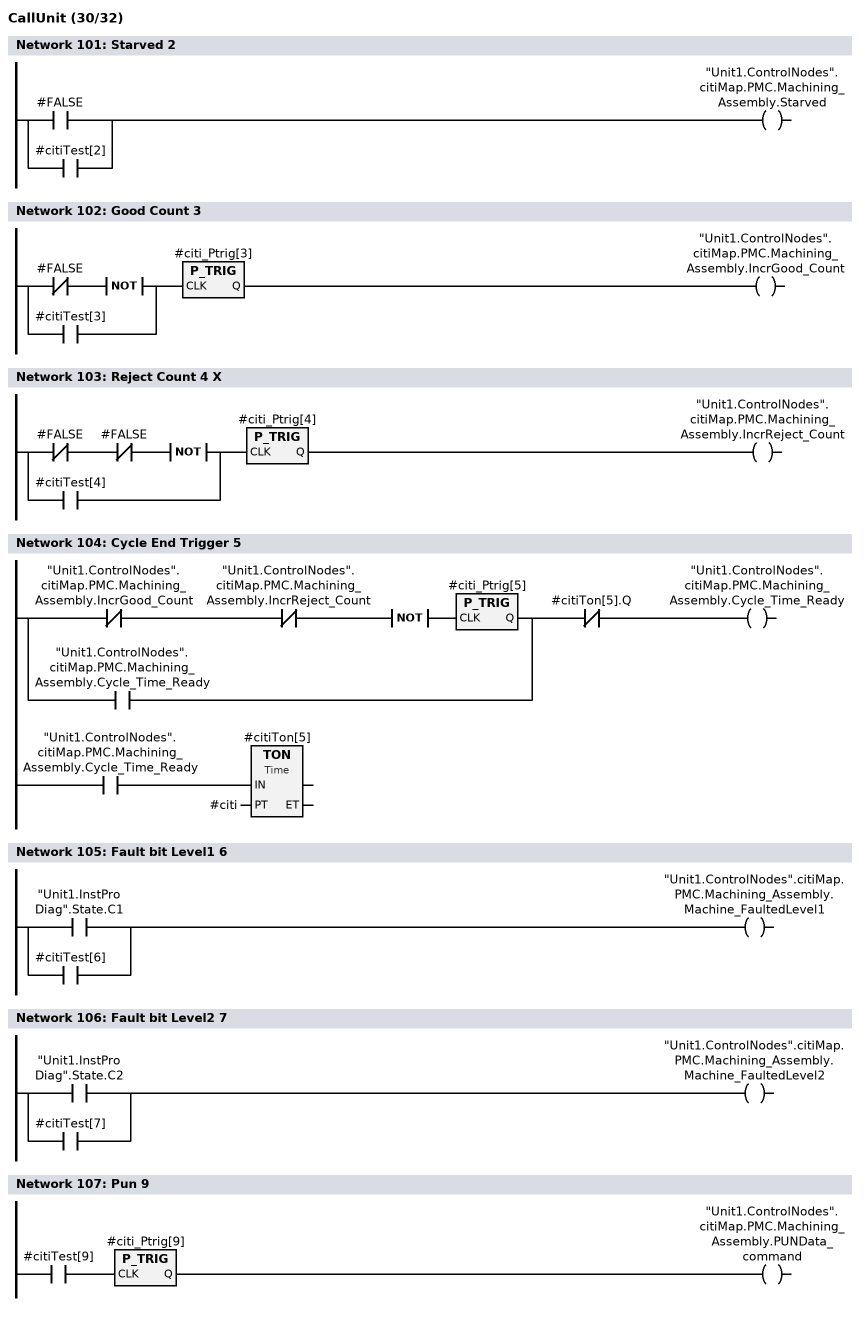
   RUNG wire#powerrail
      Contact( #FALSE )
      wire#w1
      Coil( "Unit1.ControlNodes".citiMap.PMC.Machining_Assembly.Starved )
   END_RUNG
   RUNG wire#powerrail
      Contact( #citiTest[2] )
   END_RUNG wire#w1
   // the same network as SCL:
   "Unit1.ControlNodes".citiMap.PMC.Machining_Assembly.Starved := #FALSE OR #citiTest[2];
END_REGION

REGION Network 102: Good Count 3
   RUNG wire#powerrail
      I_Contact( #FALSE )
      Not()
      wire#w1
      P_Trig( #citi_Ptrig[3] )
      Coil( "Unit1.ControlNodes".citiMap.PMC.Machining_Assembly.IncrGood_Count )
   END_RUNG
   RUNG wire#powerrail
      Contact( #citiTest[3] )
   END_RUNG wire#w1
   // the same network as SCL:
   #_w1 := NOT (NOT #FALSE) OR #citiTest[3];
   #_w2 := #_w1 AND NOT #citi_Ptrig[3];   // rising edge
   #citi_Ptrig[3] := #_w1;
   "Unit1.ControlNodes".citiMap.PMC.Machining_Assembly.IncrGood_Count := #_w2;
END_REGION

REGION Network 103: Reject Count 4 X
   RUNG wire#powerrail
      I_Contact( #FALSE )
      I_Contact( #FALSE )
      Not()
      wire#w1
      P_Trig( #citi_Ptrig[4] )
      Coil( "Unit1.ControlNodes".citiMap.PMC.Machining_Assembly.IncrReject_Count )
   END_RUNG
   RUNG wire#powerrail
      Contact( #citiTest[4] )
   END_RUNG wire#w1
   // the same network as SCL:
   #_w1 := NOT (NOT #FALSE AND NOT #FALSE) OR #citiTest[4];
   #_w2 := #_w1 AND NOT #citi_Ptrig[4];   // rising edge
   #citi_Ptrig[4] := #_w1;
   "Unit1.ControlNodes".citiMap.PMC.Machining_Assembly.IncrReject_Count := #_w2;
END_REGION

REGION Network 104: Cycle End Trigger 5
   RUNG wire#powerrail
      I_Contact( "Unit1.ControlNodes".citiMap.PMC.Machining_Assembly.IncrGood_Count )
      I_Contact( "Unit1.ControlNodes".citiMap.PMC.Machining_Assembly.IncrReject_Count )
      Not()
      P_Trig( #citi_Ptrig[5] )
      wire#w1
      I_Contact( #citiTon[5].Q )
      Coil( "Unit1.ControlNodes".citiMap.PMC.Machining_Assembly.Cycle_Time_Ready )
   END_RUNG
   RUNG wire#powerrail
      Contact( "Unit1.ControlNodes".citiMap.PMC.Machining_Assembly.Cycle_Time_Ready )
   END_RUNG wire#w1
   RUNG wire#powerrail
      Contact( "Unit1.ControlNodes".citiMap.PMC.Machining_Assembly.Cycle_Time_Ready )
      { S7_Templates := "time_type := Time" } #citiTon[5].TON(pt := #citi, et =>)
   END_RUNG
   // the same network as SCL:
   #_w1 := NOT (NOT "Unit1.ControlNodes".citiMap.PMC.Machining_Assembly.IncrGood_Count AND NOT "Unit1.ControlNodes".citiMap.PMC.Machining_Assembly.IncrReject_Count);
   #_w2 := #_w1 AND NOT #citi_Ptrig[5];   // rising edge
   #citi_Ptrig[5] := #_w1;
   "Unit1.ControlNodes".citiMap.PMC.Machining_Assembly.Cycle_Time_Ready := (#_w2 OR "Unit1.ControlNodes".citiMap.PMC.Machining_Assembly.Cycle_Time_Ready) AND NOT #citiTon[5].Q;
   #citiTon[5].TON(IN := "Unit1.ControlNodes".citiMap.PMC.Machining_Assembly.Cycle_Time_Ready, PT := #citi);
END_REGION

REGION Network 105: Fault bit Level1 6
   RUNG wire#powerrail
      Contact( "Unit1.InstProDiag".State.C1 )
      wire#w1
      Coil( "Unit1.ControlNodes".citiMap.PMC.Machining_Assembly.Machine_FaultedLevel1 )
   END_RUNG
   RUNG wire#powerrail
      Contact( #citiTest[6] )
   END_RUNG wire#w1
   // the same network as SCL:
   "Unit1.ControlNodes".citiMap.PMC.Machining_Assembly.Machine_FaultedLevel1 := "Unit1.InstProDiag".State.C1 OR #citiTest[6];
END_REGION

REGION Network 106: Fault bit Level2 7
   RUNG wire#powerrail
      Contact( "Unit1.InstProDiag".State.C2 )
      wire#w1
      Coil( "Unit1.ControlNodes".citiMap.PMC.Machining_Assembly.Machine_FaultedLevel2 )
   END_RUNG
   RUNG wire#powerrail
      Contact( #citiTest[7] )
   END_RUNG wire#w1
   // the same network as SCL:
   "Unit1.ControlNodes".citiMap.PMC.Machining_Assembly.Machine_FaultedLevel2 := "Unit1.InstProDiag".State.C2 OR #citiTest[7];
END_REGION

REGION Network 107: Pun 9
   RUNG wire#powerrail
      Contact( #citiTest[9] )
      P_Trig( #citi_Ptrig[9] )
      Coil( "Unit1.ControlNodes".citiMap.PMC.Machining_Assembly.PUNData_command )
   END_RUNG
   // the same network as SCL:
   #_w1 := #citiTest[9] AND NOT #citi_Ptrig[9];   // rising edge
   #citi_Ptrig[9] := #citiTest[9];
   "Unit1.ControlNodes".citiMap.PMC.Machining_Assembly.PUNData_command := #_w1;
END_REGION

REGION Network 108: ControlNodes.CitiMap -> Unit1. EmNodes.Andon X
END_REGION

REGION Network 109: CITI FB Cell
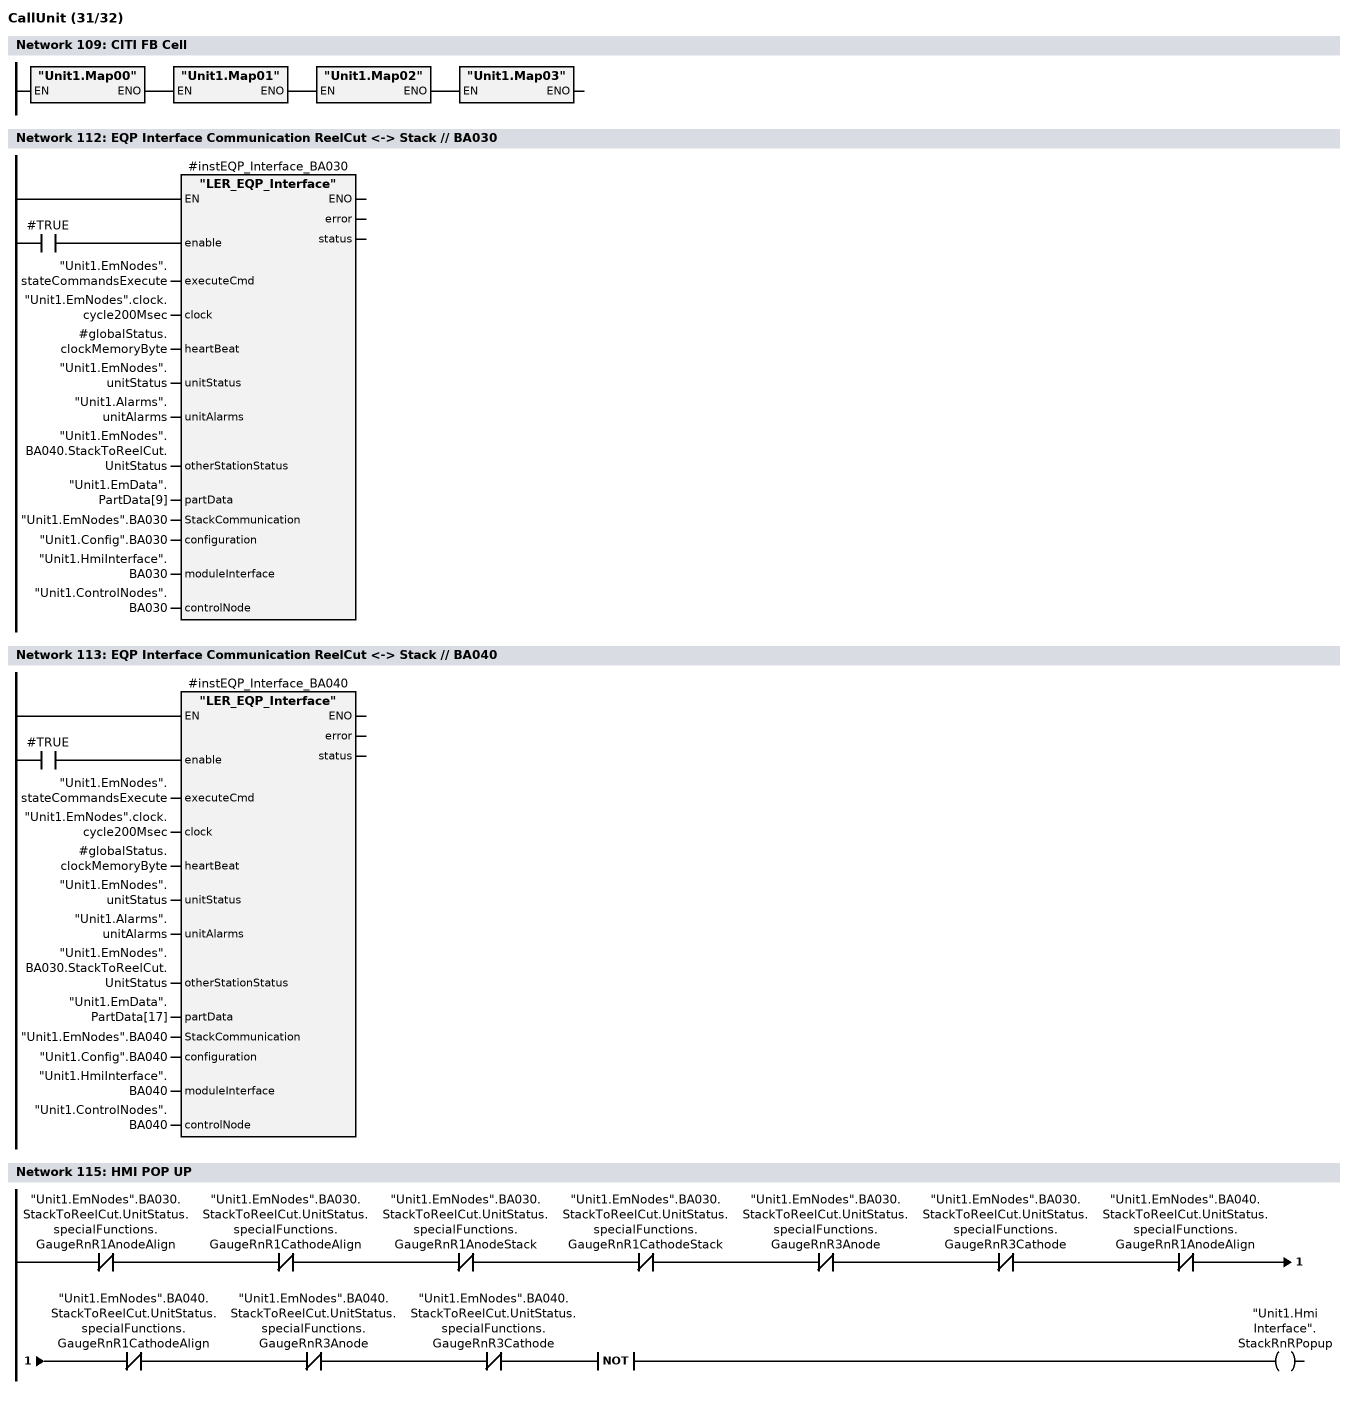
   RUNG wire#powerrail
      "Unit1.Map00"()
      "Unit1.Map01"()
      "Unit1.Map02"()
      "Unit1.Map03"()
   END_RUNG
   // the same network as SCL:
   "Unit1.Map00"(ENO => #_w1);
   "Unit1.Map01"(EN := #_w1, ENO => #_w2);
   "Unit1.Map02"(EN := #_w2, ENO => #_w3);
   IF #_w3 THEN "Unit1.Map03"(); END_IF;
END_REGION

REGION Network 111: ******************** PLC Communication ********************
END_REGION

REGION Network 112: EQP Interface Communication ReelCut <-> Stack // BA030
   RUNG wire#powerrail
      #instEQP_Interface_BA030(enable := wire#w1, executeCmd := "Unit1.EmNodes".stateCommandsExecute, clock := "Unit1.EmNodes".clock.cycle200Msec, heartBeat := #globalStatus.clockMemoryByte, unitStatus := "Unit1.EmNodes".unitStatus, unitAlarms := "Unit1.Alarms".unitAlarms, otherStationStatus := "Unit1.EmNodes".BA040.StackToReelCut.UnitStatus, partData := "Unit1.EmData".PartData[9], StackCommunication := "Unit1.EmNodes".BA030, configuration := "Unit1.Config".BA030, moduleInterface := "Unit1.HmiInterface".BA030, controlNode := "Unit1.ControlNodes".BA030, error =>, status =>)
   END_RUNG
   RUNG wire#powerrail
      Contact( #TRUE )
   END_RUNG wire#w1
   // the same network as SCL:
   #instEQP_Interface_BA030(enable := #TRUE,   // "LER_EQP_Interface"
                           executeCmd := "Unit1.EmNodes".stateCommandsExecute,
                           clock := "Unit1.EmNodes".clock.cycle200Msec,
                           heartBeat := #globalStatus.clockMemoryByte,
                           unitStatus := "Unit1.EmNodes".unitStatus,
                           unitAlarms := "Unit1.Alarms".unitAlarms,
                           otherStationStatus := "Unit1.EmNodes".BA040.StackToReelCut.UnitStatus,
                           partData := "Unit1.EmData".PartData[9],
                           StackCommunication := "Unit1.EmNodes".BA030,
                           configuration := "Unit1.Config".BA030,
                           moduleInterface := "Unit1.HmiInterface".BA030,
                           controlNode := "Unit1.ControlNodes".BA030);
END_REGION

REGION Network 113: EQP Interface Communication ReelCut <-> Stack // BA040
   RUNG wire#powerrail
      #instEQP_Interface_BA040(enable := wire#w1, executeCmd := "Unit1.EmNodes".stateCommandsExecute, clock := "Unit1.EmNodes".clock.cycle200Msec, heartBeat := #globalStatus.clockMemoryByte, unitStatus := "Unit1.EmNodes".unitStatus, unitAlarms := "Unit1.Alarms".unitAlarms, otherStationStatus := "Unit1.EmNodes".BA030.StackToReelCut.UnitStatus, partData := "Unit1.EmData".PartData[17], StackCommunication := "Unit1.EmNodes".BA040, configuration := "Unit1.Config".BA040, moduleInterface := "Unit1.HmiInterface".BA040, controlNode := "Unit1.ControlNodes".BA040, error =>, status =>)
   END_RUNG
   RUNG wire#powerrail
      Contact( #TRUE )
   END_RUNG wire#w1
   // the same network as SCL:
   #instEQP_Interface_BA040(enable := #TRUE,   // "LER_EQP_Interface"
                           executeCmd := "Unit1.EmNodes".stateCommandsExecute,
                           clock := "Unit1.EmNodes".clock.cycle200Msec,
                           heartBeat := #globalStatus.clockMemoryByte,
                           unitStatus := "Unit1.EmNodes".unitStatus,
                           unitAlarms := "Unit1.Alarms".unitAlarms,
                           otherStationStatus := "Unit1.EmNodes".BA030.StackToReelCut.UnitStatus,
                           partData := "Unit1.EmData".PartData[17],
                           StackCommunication := "Unit1.EmNodes".BA040,
                           configuration := "Unit1.Config".BA040,
                           moduleInterface := "Unit1.HmiInterface".BA040,
                           controlNode := "Unit1.ControlNodes".BA040);
END_REGION

REGION Network 114: ******************** Stack RnR Mode POP UP ********************
END_REGION

REGION Network 115: HMI POP UP
   RUNG wire#powerrail
      I_Contact( "Unit1.EmNodes".BA030.StackToReelCut.UnitStatus.specialFunctions.GaugeRnR1AnodeAlign )
      I_Contact( "Unit1.EmNodes".BA030.StackToReelCut.UnitStatus.specialFunctions.GaugeRnR1CathodeAlign )
      I_Contact( "Unit1.EmNodes".BA030.StackToReelCut.UnitStatus.specialFunctions.GaugeRnR1AnodeStack )
      I_Contact( "Unit1.EmNodes".BA030.StackToReelCut.UnitStatus.specialFunctions.GaugeRnR1CathodeStack )
      I_Contact( "Unit1.EmNodes".BA030.StackToReelCut.UnitStatus.specialFunctions.GaugeRnR3Anode )
      I_Contact( "Unit1.EmNodes".BA030.StackToReelCut.UnitStatus.specialFunctions.GaugeRnR3Cathode )
      I_Contact( "Unit1.EmNodes".BA040.StackToReelCut.UnitStatus.specialFunctions.GaugeRnR1AnodeAlign )
      I_Contact( "Unit1.EmNodes".BA040.StackToReelCut.UnitStatus.specialFunctions.GaugeRnR1CathodeAlign )
      I_Contact( "Unit1.EmNodes".BA040.StackToReelCut.UnitStatus.specialFunctions.GaugeRnR3Anode )
      I_Contact( "Unit1.EmNodes".BA040.StackToReelCut.UnitStatus.specialFunctions.GaugeRnR3Cathode )
      Not()
      Coil( "Unit1.HmiInterface".StackRnRPopup )
   END_RUNG
   // the same network as SCL:
   "Unit1.HmiInterface".StackRnRPopup := NOT (NOT "Unit1.EmNodes".BA030.StackToReelCut.UnitStatus.specialFunctions.GaugeRnR1AnodeAlign AND NOT "Unit1.EmNodes".BA030.StackToReelCut.UnitStatus.specialFunctions.GaugeRnR1CathodeAlign AND NOT "Unit1.EmNodes".BA030.StackToReelCut.UnitStatus.specialFunctions.GaugeRnR1AnodeStack AND NOT "Unit1.EmNodes".BA030.StackToReelCut.UnitStatus.specialFunctions.GaugeRnR1CathodeStack AND NOT "Unit1.EmNodes".BA030.StackToReelCut.UnitStatus.specialFunctions.GaugeRnR3Anode AND NOT "Unit1.EmNodes".BA030.StackToReelCut.UnitStatus.specialFunctions.GaugeRnR3Cathode AND NOT "Unit1.EmNodes".BA040.StackToReelCut.UnitStatus.specialFunctions.GaugeRnR1AnodeAlign AND NOT "Unit1.EmNodes".BA040.StackToReelCut.UnitStatus.specialFunctions.GaugeRnR1CathodeAlign AND NOT "Unit1.EmNodes".BA040.StackToReelCut.UnitStatus.specialFunctions.GaugeRnR3Anode AND NOT "Unit1.EmNodes".BA040.StackToReelCut.UnitStatus.specialFunctions.GaugeRnR3Cathode);
END_REGION

REGION Network 116: Radius Value To Safety
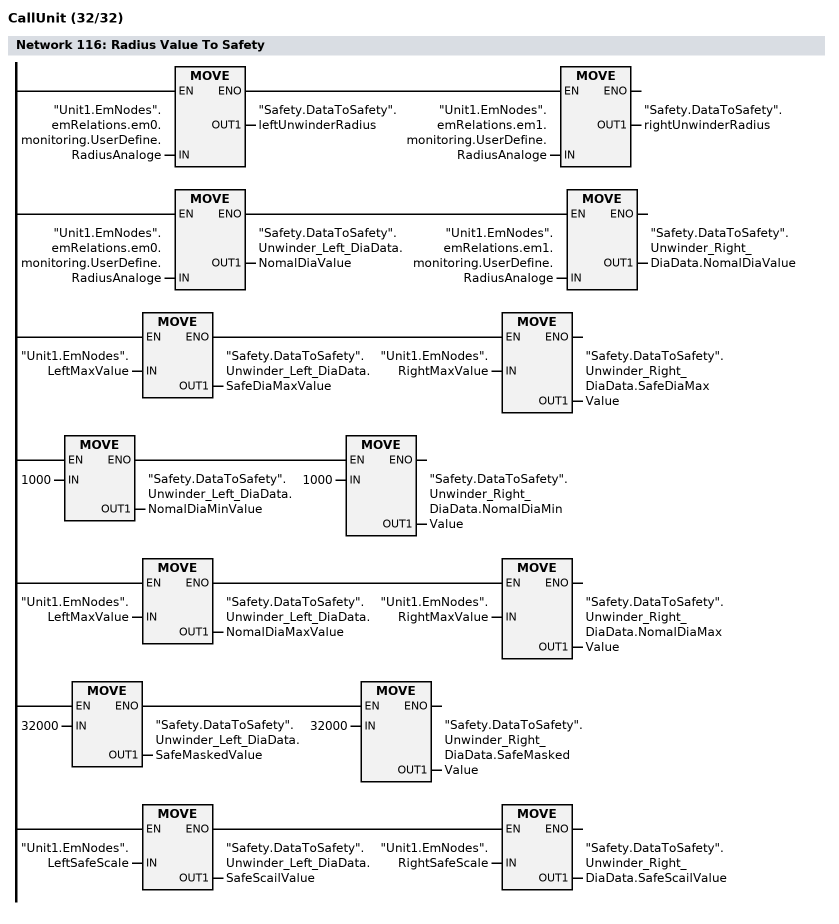
   RUNG wire#powerrail
      Move(in := "Unit1.EmNodes".emRelations.em0.monitoring.UserDefine.RadiusAnaloge, out1 => "Safety.DataToSafety".leftUnwinderRadius)
      Move(in := "Unit1.EmNodes".emRelations.em1.monitoring.UserDefine.RadiusAnaloge, out1 => "Safety.DataToSafety".rightUnwinderRadius)
   END_RUNG
   RUNG wire#powerrail
      Move(in := "Unit1.EmNodes".emRelations.em0.monitoring.UserDefine.RadiusAnaloge, out1 => "Safety.DataToSafety".Unwinder_Left_DiaData.NomalDiaValue)
      Move(in := "Unit1.EmNodes".emRelations.em1.monitoring.UserDefine.RadiusAnaloge, out1 => "Safety.DataToSafety".Unwinder_Right_DiaData.NomalDiaValue)
   END_RUNG
   RUNG wire#powerrail
      Move(in := "Unit1.EmNodes".LeftMaxValue, out1 => "Safety.DataToSafety".Unwinder_Left_DiaData.SafeDiaMaxValue)
      Move(in := "Unit1.EmNodes".RightMaxValue, out1 => "Safety.DataToSafety".Unwinder_Right_DiaData.SafeDiaMaxValue)
   END_RUNG
   RUNG wire#powerrail
      Move(in := 1000, out1 => "Safety.DataToSafety".Unwinder_Left_DiaData.NomalDiaMinValue)
      Move(in := 1000, out1 => "Safety.DataToSafety".Unwinder_Right_DiaData.NomalDiaMinValue)
   END_RUNG
   RUNG wire#powerrail
      Move(in := "Unit1.EmNodes".LeftMaxValue, out1 => "Safety.DataToSafety".Unwinder_Left_DiaData.NomalDiaMaxValue)
      Move(in := "Unit1.EmNodes".RightMaxValue, out1 => "Safety.DataToSafety".Unwinder_Right_DiaData.NomalDiaMaxValue)
   END_RUNG
   RUNG wire#powerrail
      Move(in := 32000, out1 => "Safety.DataToSafety".Unwinder_Left_DiaData.SafeMaskedValue)
      Move(in := 32000, out1 => "Safety.DataToSafety".Unwinder_Right_DiaData.SafeMaskedValue)
   END_RUNG
   RUNG wire#powerrail
      Move(in := "Unit1.EmNodes".LeftSafeScale, out1 => "Safety.DataToSafety".Unwinder_Left_DiaData.SafeScailValue)
      Move(in := "Unit1.EmNodes".RightSafeScale, out1 => "Safety.DataToSafety".Unwinder_Right_DiaData.SafeScailValue)
   END_RUNG
   // the same network as SCL:
   "Safety.DataToSafety".leftUnwinderRadius := "Unit1.EmNodes".emRelations.em0.monitoring.UserDefine.RadiusAnaloge;
   "Safety.DataToSafety".rightUnwinderRadius := "Unit1.EmNodes".emRelations.em1.monitoring.UserDefine.RadiusAnaloge;
   "Safety.DataToSafety".Unwinder_Left_DiaData.NomalDiaValue := "Unit1.EmNodes".emRelations.em0.monitoring.UserDefine.RadiusAnaloge;
   "Safety.DataToSafety".Unwinder_Right_DiaData.NomalDiaValue := "Unit1.EmNodes".emRelations.em1.monitoring.UserDefine.RadiusAnaloge;
   "Safety.DataToSafety".Unwinder_Left_DiaData.SafeDiaMaxValue := "Unit1.EmNodes".LeftMaxValue;
   "Safety.DataToSafety".Unwinder_Right_DiaData.SafeDiaMaxValue := "Unit1.EmNodes".RightMaxValue;
   "Safety.DataToSafety".Unwinder_Left_DiaData.NomalDiaMinValue := 1000;
   "Safety.DataToSafety".Unwinder_Right_DiaData.NomalDiaMinValue := 1000;
   "Safety.DataToSafety".Unwinder_Left_DiaData.NomalDiaMaxValue := "Unit1.EmNodes".LeftMaxValue;
   "Safety.DataToSafety".Unwinder_Right_DiaData.NomalDiaMaxValue := "Unit1.EmNodes".RightMaxValue;
   "Safety.DataToSafety".Unwinder_Left_DiaData.SafeMaskedValue := 32000;
   "Safety.DataToSafety".Unwinder_Right_DiaData.SafeMaskedValue := 32000;
   "Safety.DataToSafety".Unwinder_Left_DiaData.SafeScailValue := "Unit1.EmNodes".LeftSafeScale;
   "Safety.DataToSafety".Unwinder_Right_DiaData.SafeScailValue := "Unit1.EmNodes".RightSafeScale;
END_REGION
END_FUNCTION_BLOCK
